TYPE UDT 19
VERSION : 0.0
  STRUCT
   A_SCLight : BOOL ;	//Screen light
   A_SCDark : BOOL ;	//Screen darkening
   A_KeyDisable : BOOL ;	//Key disable
   A_ClearCanAl : BOOL ;	//Clear cancel alarms
   A_ClearRecAl : BOOL ;	//Clear recall alarms
   f0_5 : BOOL ;
   f0_6 : BOOL ;
   A_ActWCS : BOOL ;	//Actual value in WCS 0=MCS
   A_PLCExtViewerReject : BOOL ;	//External viewer reject
   A_PLCExtViewerMode : BOOL ;	//External viewer mode
   f1_2 : BOOL ;
   f1_3 : BOOL ;
   f1_4 : BOOL ;
   f1_5 : BOOL ;
   f1_6 : BOOL ;
   f1_7 : BOOL ;
   A_1stError1 : WORD ;	//1st error HIGRAPH
   A_1stError2 : WORD ;	//1st error HIGRAPH
   A_ASpi1percent : BYTE ;	//Analog spindle 1:
   A_ASpi2percent : BYTE ;
   A_MCPChan : BYTE ;
   A_OEM1 : BOOL ;
   A_OEM2 : BOOL ;
   A_AToolMeas : BOOL ;	//AutoToolMeasure
   f9_3 : BOOL ;
   f9_4 : BOOL ;
   f9_5 : BOOL ;
   f9_6 : BOOL ;
   f9_7 : BOOL ;
   A_Hardkey : BYTE ;	//PLC Hardkeys
   f11 : BYTE ;	//Reserved for hardkeys
   f12_0 : BOOL ;
   f12_1 : BOOL ;
   A_COM2 : BOOL ;
   A_COM1 : BOOL ;
   A_V24stop : BOOL ;
   A_V24ext : BOOL ;
   A_V24off : BOOL ;
   A_V24on : BOOL ;
   A_TeachDisable : BOOL ;
   f13_1 : BOOL ;
   f13_2 : BOOL ;
   f13_3 : BOOL ;
   f13_4 : BOOL ;
   A_PPdeload : BOOL ;
   A_PPload : BOOL ;
   A_PPsel : BOOL ;
   A_V24Index1 : BYTE ;
   A_V24Index2 : BYTE ;
   A_V24NoFile1 : BYTE ;
   A_V24NoFile2 : BYTE ;
   A_res18 : BYTE ;
   A_res19 : BYTE ;	//Message counter
   f20_0 : BOOL ;
   E_SCDark : BOOL ;	//Screen darkening
   E_Cancel : BOOL ;	//Cancel
   E_CanCleared : BOOL ;	//Cancel alarms cleared
   E_RecCleared : BOOL ;	//Recall alarms cleared
   f20_5 : BOOL ;	//res. Language
   E_SimActiv : BOOL ;	//Simulation active
   E_ActWCS : BOOL ;	//Switchover MCS/WCS 0=MCS
   E_ActivWA : BYTE ;
   E_Chan : BYTE ;	//Channel displayed
   f23 : BYTE ;
   E_V24Err : BOOL ;
   E_V24OK : BOOL ;
   E_V24COM2 : BOOL ;
   E_V24COM1 : BOOL ;
   E_V24stop : BOOL ;
   E_V24ext : BOOL ;
   E_V24off : BOOL ;
   E_V24on : BOOL ;
   E_V24Error : BYTE ;	//V24: Error Byte
   E_res26_0 : BOOL ;	//Reserved
   E_PPOK : BOOL ;	//Part program status OK
   E_PPErr : BOOL ;	//Part program status Error
   E_PPAct : BOOL ;	//Part program status active
   f26_4 : BOOL ;	//Reserved
   E_PPdeload : BOOL ;	//Part program status deloading
   E_PPload : BOOL ;	//Part program status loading
   E_PPsel : BOOL ;	//Part program status selecting
   E_PPError : BYTE ;	//Part program status Error
   A_PictNo : INT ;
   A_PictOn : BOOL ;
   A_PictOff : BOOL ;
   f30_2 : BOOL ;
   f30_3 : BOOL ;
   f30_4 : BOOL ;
   f30_5 : BOOL ;
   f30_6 : BOOL ;
   f30_7 : BOOL ;
   E_PictOK : BOOL ;
   E_PictOn : BOOL ;
   E_PictAct : BOOL ;
   E_PictOff : BOOL ;
   E_PictErr : BOOL ;
   f31_5 : BOOL ;
   f31_6 : BOOL ;
   E_NotAct : BOOL ;
   A_FuncNo : BYTE ;
   A_Par1 : BYTE ;
   A_Par2 : BYTE ;
   A_Par3 : BYTE ;
   E_FuncErr : BYTE ;
   f37 : BYTE ;
   f38 : BYTE ;
   f39 : BYTE ;
   res40 : ARRAY  [0 .. 9 ] OF BYTE ;
   MMC2 : STRUCT
    A_SCLight : BOOL ;	//Screen light
    A_SCDark : BOOL ;	//Screen darkening
    A_KeyDisable : BOOL ;	//Key disable
    A_ClearCanAl : BOOL ;	//Clear cancel alarms
    A_ClearRecAl : BOOL ;	//Clear recall alarms
    f0_5 : BOOL ;
    f0_6 : BOOL ;
    A_ActWCS : BOOL ;	//Actual value in WCS 0=MCS
    A_1stError1 : WORD ;	//1st error HIGRAPH
    A_1stError2 : WORD ;	//1st error HIGRAPH
    A_ASpi1percent : BYTE ;	//Analog spindle 1:
    A_ASpi2percent : BYTE ;
    A_MCPChan : BYTE ;
    A_OEM1 : BOOL ;
    A_OEM2 : BOOL ;
    A_AToolMeas : BOOL ;	//AutoToolMeasure
    f9_3 : BOOL ;
    f9_4 : BOOL ;
    f9_5 : BOOL ;
    f9_6 : BOOL ;
    f9_7 : BOOL ;
    A_Hardkey : BYTE ;	//PLC Hardkeys
    f11 : BYTE ;	//Reserved for hardkeys
    f12_0 : BOOL ;
    f12_1 : BOOL ;
    A_COM2 : BOOL ;
    A_COM1 : BOOL ;
    A_V24stop : BOOL ;
    A_V24ext : BOOL ;
    A_V24off : BOOL ;
    A_V24on : BOOL ;
    f13_0 : BOOL ;
    f13_1 : BOOL ;
    f13_2 : BOOL ;
    f13_3 : BOOL ;
    f13_4 : BOOL ;
    A_PPdeload : BOOL ;
    A_PPload : BOOL ;
    A_PPsel : BOOL ;
    A_V24Index1 : BYTE ;
    A_V24Index2 : BYTE ;
    A_V24NoFile1 : BYTE ;
    A_V24NoFile2 : BYTE ;
    A_res18 : BYTE ;
    A_res19 : BYTE ;	//Message counter
    f20_0 : BOOL ;
    E_SCDark : BOOL ;	//Screen darkening
    E_Cancel : BOOL ;	//Cancel
    E_CanCleared : BOOL ;	//Cancel alarms cleared
    E_RecCleared : BOOL ;	//Recall alarms cleared
    f20_5 : BOOL ;	//res. Language
    E_SimActiv : BOOL ;	//Simulation active
    E_ActWCS : BOOL ;	//Switchover MCS/WCS 0=MCS
    E_ActivWA : BYTE ;
    E_Chan : BYTE ;	//Channel displayed
    f23 : BYTE ;
    E_V24Err : BOOL ;
    E_V24OK : BOOL ;
    E_V24COM2 : BOOL ;
    E_V24COM1 : BOOL ;
    E_V24stop : BOOL ;
    E_V24ext : BOOL ;
    E_V24off : BOOL ;
    E_V24on : BOOL ;
    E_V24Error : BYTE ;	//V24: Error Byte
    E_res26_0 : BOOL ;	//Reserved
    E_PPOK : BOOL ;	//Part program status OK
    E_PPErr : BOOL ;	//Part program status Error
    E_PPAct : BOOL ;	//Part program status active
    f26_4 : BOOL ;	//Reserved
    E_PPdeload : BOOL ;	//Part program status deloading
    E_PPload : BOOL ;	//Part program status loading
    E_PPsel : BOOL ;	//Part program status selecting
    E_PPError : BYTE ;	//Part program status Error
    A_PictNo : INT ;
    A_PictOn : BOOL ;
    A_PictOff : BOOL ;
    f30_2 : BOOL ;
    f30_3 : BOOL ;
    f30_4 : BOOL ;
    f30_5 : BOOL ;
    f30_6 : BOOL ;
    f30_7 : BOOL ;
    E_PictOK : BOOL ;
    E_PictOn : BOOL ;
    E_PictAct : BOOL ;
    E_PictOff : BOOL ;
    E_PictErr : BOOL ;
    f31_5 : BOOL ;
    f31_6 : BOOL ;
    E_NotAct : BOOL ;
    A_FuncNo : BYTE ;
    A_Par1 : BYTE ;
    A_Par2 : BYTE ;
    A_Par3 : BYTE ;
    E_FuncErr : BYTE ;
    f37 : BYTE ;
    f38 : BYTE ;
    f39 : BYTE ;
    res40 : ARRAY  [0 .. 9 ] OF BYTE ;
   END_STRUCT ;	//M to N
   ONL_REQUEST : WORD ;
   ONL_CONFIRM : WORD ;
   PAR_CLIENT_IDENT : WORD ;
   PAR_MMC_TYP : BYTE ;
   PAR_MSTT_ADR : BYTE ;
   PAR_STATUS : BYTE ;
   PAR_Z_INFO : BYTE ;
   MtoNAlive : WORD ;
   f112 : BYTE ;
   ParOpKeyAdr : BYTE ;
   ParTcuIndex : BYTE ;
   f115 : BYTE ;
   Tcu1KeyAdr : BYTE ;
   Tcu2KeyAdr : BYTE ;
   Tcu1Index : BYTE ;
   Tcu2Index : BYTE ;
   MMC1_CLIENT_IDENT : WORD ;
   MMC1_TYP : BYTE ;
   MMC1_MSTT_ADR : BYTE ;
   MMC1_STATUS : BYTE ;
   MMC1_Z_INFO : BYTE ;
   MMC1_SHIFT_LOCK : BOOL ;
   MMC1_MSTT_SHIFT_LOCK : BOOL ;
   MMC1_ACTIVE_REQ : BOOL ;
   MMC1_ACTIVE_PERM : BOOL ;
   MMC1_ACTIVE_CHANGED : BOOL ;
   MMC1_CHANGED_DENIED : BOOL ;
   MMC1_TCU_SHIFT_LOCK : BOOL ;
   f127 : BYTE ;
   MMC1_TRANS_DB : WORD ;
   MMC2_CLIENT_IDENT : WORD ;
   MMC2_TYP : BYTE ;
   MMC2_MSTT_ADR : BYTE ;
   MMC2_STATUS : BYTE ;
   MMC2_Z_INFO : BYTE ;
   MMC2_SHIFT_LOCK : BOOL ;
   MMC2_MSTT_SHIFT_LOCK : BOOL ;
   MMC2_ACTIVE_REQ : BOOL ;
   MMC2_ACTIVE_PERM : BOOL ;
   MMC2_ACTIVE_CHANGED : BOOL ;
   MMC2_CHANGED_DENIED : BOOL ;
   MMC2_TCU_SHIFT_LOCK : BOOL ;
   f137 : BYTE ;
   MMC2_TRANS_DB : WORD ;
   A_Subtype : INT ;	//for Codecarrier Input from PLC
   A_Duplo : INT ;
   A_Ident : STRING  [32 ];
   A_Tnumber : INT ;
   A_MagazinePlace : INT ;
   A_MagazinePlaceType : INT ;
   A_ToolSize_Upper : BYTE ;
   A_ToolSize_Down : BYTE ;
   A_ToolSize_Left : BYTE ;
   A_ToolSize_Right : BYTE ;
   A_Channel : BYTE ;
   A_LoadingPlace : BYTE ;
   A_Magazine : INT ;
   A_Unit : BYTE ;
   A_NCU_Index : BYTE ;
   A_FileIndex : INT ;
   A_ActiveEnable : BOOL ;
   A_Override : BOOL ;
   A_LoadTool : BOOL ;
   A_DeleteTool : BOOL ;
   E_Subtype : INT ;	//for Codecarrier Output to PLC
   E_Duplo : INT ;
   E_Ident : STRING  [32 ];
   E_Tnumber : INT ;
   E_ToolState : INT ;
   E_MagazinePlaceType : INT ;
   E_ToolSize_Upper : BYTE ;
   E_ToolSize_Down : BYTE ;
   E_ToolSize_Left : BYTE ;
   E_ToolSize_Right : BYTE ;
   E_Magazine : INT ;
   E_MagazinePlace : INT ;
   A_ReqMMC1 : BOOL ;	//for Codecarrier Request MMC-Interface1
   A_ReqMMC2 : BOOL ;	//for Codecarrier Request MMC-Interface2
   A_K_Code : BYTE ;
   E_Done : BOOL ;
   E_Error : BOOL ;
   E_Active : BOOL ;	// CodeCarrierReadEnable : BOOL;
// CodeCarrierWriteEnable : BOOL;
   E_K_CodeError : BYTE ;	//Identify for Error_Code
   E_Error_Code : INT ;
   E_Req : BOOL ;	//for Positioning
   f257 : BYTE ;
   A_Done : BOOL ;
   A_Error : BOOL ;
   A_Active : BOOL ;
   f258_3 : BOOL ;
   f258_4 : BOOL ;
   f258_5 : BOOL ;
   f258_6 : BOOL ;
   f258_7 : BOOL ;
   E_TDC_Read : BOOL ;
   E_TDC_Write : BOOL ;
   E_TDC_Cancel : BOOL ;
   A_Error_Code : INT ;
   E_PMagazine : INT ;
   E_PMagazinePlace : INT ;
   E_PTnumber : INT ;	//TPM-Data
   A_TPMStatus : INT ;
   A_TPMCounter : ARRAY  [1 .. 32 ] OF DINT ;
   A_HWeelSimOvr : BYTE ;
   f399 : BYTE ;
   A_SimOvr : INT ;
  END_STRUCT ;	
END_TYPE

TYPE UDT 21
VERSION : 0.0
  STRUCT
   f0_0 : BOOL ;
   f0_1 : BOOL ;
   f0_2 : BOOL ;
   A_DRF : BOOL ;	//Activate DRF
   A_SBL : BOOL ;	//Activate single block
   A_M01 : BOOL ;	//Activate M01
   A_DRY : BOOL ;	//Activate dry run feedrate
   f0_7 : BOOL ;
   A_Ref : BOOL ;	//Activate referencing
   A_ProtZone : BOOL ;	//Enable protection zones
   A_SynOff : BOOL ;	//Synchronous action off
   A_TM_TimOut : BOOL ;	//Activate time-out (TM)
   A_CLC_Stop : BOOL ;	//CLC stop
   A_CLC_OR : BOOL ;	//CLC override
   A_PLC_ActCompl : BOOL ;	//PLC action complete
   A_ProgTest : BOOL ;	//Activate program test
   A_SKP0 : BOOL ;	//Activate skip block \0
   A_SKP1 : BOOL ;	//Activate skip block \1
   A_SKP2 : BOOL ;	//Activate skip block \2
   A_SKP3 : BOOL ;	//Activate skip block \3
   A_SKP4 : BOOL ;	//Activate skip block \4
   A_SKP5 : BOOL ;	//Activate skip block \5
   A_SKP6 : BOOL ;	//Activate skip block \6
   A_SKP7 : BOOL ;	//Activate skip block \7
   A_StrokEnab : BOOL ;	//Stroke enable
   A_ManStrokEnab : BOOL ;	//Manual stroke enable
   A_StrokSup : BOOL ;	//Stroke suppression
   A_StrokDelayed : BOOL ;	//Stroke delayed
   A_StrokStop : BOOL ;	//Stroke not operating
   A_ManRelStroke2 : BOOL ;	// Manual release of stroke 2
   A3_6 : BOOL ;
   A3_7 : BOOL ;
   A_FD_OR : BYTE ;	//Feedrate override
   A_RT_OR : BYTE ;	//Rapid traverse override
   A_FDdisable : BOOL ;	//Feed disable
   A_RIdisable : BOOL ;	//Read-in disable
   A_DeleteDTG : BOOL ;	//Delete distance to go
   A_SP_Clear : BOOL ;	//Clear SP repetitions
   A_ProgAbort : BOOL ;	//Program level abort
   A_F_Limit : BOOL ;	//Tool path feedrate limitation
   A_RT_ORA : BOOL ;	//Rapid traverse override active
   A_FD_ORA : BOOL ;	//Feedrate override active
   A_NCStartDisabl : BOOL ;	//NC start disable
   A_NCStart : BOOL ;	//NC start
   A_NCStopBlock : BOOL ;	//NC stop at block limit
   A_NCStop : BOOL ;	//NC stop
   A_NCStopASp : BOOL ;	//NC stop axes plus spindle
   A_SuppStartLock : BOOL ;	// Suppress Start Lock
   f7_6 : BOOL ;
   A_Reset : BOOL ;	//Reset
   A_MRP : ARRAY  [1 .. 10 ] OF BOOL ;	//Activate machine-related protection area [1..10]
   A_CSP : ARRAY  [1 .. 10 ] OF BOOL ;	//Activate channel-specific protection area [1..10]
   A_Geo : ARRAY  [1 .. 3 ] OF STRUCT 	//Control signals for geometry axis [1..3]
    HW1 : BOOL ;	//Activate handwheel 1
    HW2 : BOOL ;	//Activate handwheel 2
    HW3 : BOOL ;	//Activate handwheel 3
    FDStop : BOOL ;	//Feed stop
    Disabl : BOOL ;	//Traversing key disable
    RapidTrOR : BOOL ;	//Rapid traverse override
    Minus : BOOL ;	//Traversing key minus
    Plus : BOOL ;	//Traversing key plus
    INC1 : BOOL ;	//INC 1
    INC10 : BOOL ;	//INC 10
    INC100 : BOOL ;	//INC 100
    INC1000 : BOOL ;	//INC 1000
    INC10000 : BOOL ;	//INC 10000
    INCVar : BOOL ;	//INC variable
    OEM : BYTE ;	//OEM signals
    InvHWDirOfRot : BOOL ;	// Inverting handwheel direction of rotation
    f3_1 : BOOL ;
    f3_2 : BOOL ;
    f3_3 : BOOL ;
    f3_4 : BOOL ;
    f3_5 : BOOL ;
    f3_6 : BOOL ;
    f3_7 : BOOL ;
   END_STRUCT ;
   f24_0 : BOOL ;
   f24_1 : BOOL ;
   f24_2 : BOOL ;
   E_MMC_DRF : BOOL ;	//MMC DRF selected
   f24_4 : BOOL ;
   E_MMC_M01 : BOOL ;	//MMC M01 selected
   E_MMC_DRY : BOOL ;	//MMC Dry run feedrate selected
   f24_7 : BOOL ;
   E_MMC_REPOSPM_0 : BOOL ;	//MMC REPOSPATHMODE 0
   E_MMC_REPOSPM_1 : BOOL ;	//MMC REPOSPATHMODE 1
   E_MMC_REPOSPM_2 : BOOL ;	//MMC REPOSPATHMODE 2
   E_MMC_FD_OR4RT_OR : BOOL ;	//MMC Feedrate override for rapid traverse selected
   E_MMC_REPOSMode : BOOL ;	//MMC REPOS MODE EDGE
   f25_5 : BOOL ;
   f25_6 : BOOL ;
   E_MMC_ProgTest : BOOL ;	//Program test selected
   E_MMC_SKP0 : BOOL ;	//MMC skip block selected \0
   E_MMC_SKP1 : BOOL ;	//MMC skip block selected \1
   E_MMC_SKP2 : BOOL ;	//MMC skip block selected \2
   E_MMC_SKP3 : BOOL ;	//MMC skip block selected \3
   E_MMC_SKP4 : BOOL ;	//MMC skip block selected \4
   E_MMC_SKP5 : BOOL ;	//MMC skip block selected \5
   E_MMC_SKP6 : BOOL ;	//MMC skip block selected \6
   E_MMC_SKP7 : BOOL ;	//MMC skip block selected \7
   E_MMC_SKP8 : BOOL ;	//MMC skip block selected \8
   E_MMC_SKP9 : BOOL ;	//MMC skip block selected \9
   f27_2 : BOOL ;
   f27_3 : BOOL ;
   f27_4 : BOOL ;
   f27_5 : BOOL ;
   f27_6 : BOOL ;
   f27_7 : BOOL ;
   A_OEM : BYTE ;
   A_FixedFD1 : BOOL ;	//Fixed feeds
   A_FixedFD2 : BOOL ;
   A_FixedFD3 : BOOL ;
   A_FixedFD4 : BOOL ;
   A_PTP_Travel : BOOL ;	//Activate PTP travel
   A_DisablWP_Counter : BOOL ;	//Disable workpiece counter
   A_DisablWearMon : BOOL ;	//Disable wear monitoring
   A_DontDisablTool : BOOL ;	//Do not disable tool
   A_ContHW1 : BOOL ;	//Activate contour handwheels
   A_ContHW2 : BOOL ;
   A_ContHW3 : BOOL ;
   A_ContHWsim : BOOL ;	//Simulated contour handwheel on
   A_ContHWneg : BOOL ;	//Contour handwheel neg. route
   A_NCKrelatedM01 : BOOL ;	// Activate NCK-related M01
   f30_6 : BOOL ;
   A_NoToolChangeCmd : BOOL ;	// No tool change commands
   A_REPOSPM_0 : BOOL ;	//REPOSPATHMODE 0
   A_REPOSPM_1 : BOOL ;	//REPOSPATHMODE 1
   A_REPOSPM_2 : BOOL ;	//REPOSPATHMODE 2
   f31_3 : BOOL ;
   A_REPOSMode : BOOL ;	//REPOS MODE EDGE
   A_InvCHWDirOfRot : BOOL ;	// Inverting contour handwheel direction of rotation
   A_SKP8 : BOOL ;	//Activate skip block \8
   A_SKP9 : BOOL ;	//Activate skip block \9
   E_ExecExtern : BOOL ;	//Execution from external source active
   f32_1 : BOOL ;
   f32_2 : BOOL ;
   E_ActBlock : BOOL ;	//Action block active
   E_BegBlock : BOOL ;	//Approach block active
   E_M01 : BOOL ;	//M0/M1 active
   E_LastActBlock : BOOL ;	//Last action block active
   f32_7 : BOOL ;
   E_Ref : BOOL ;	//Referencing active
   E_OrieToolholder : BOOL ;	// Orientable toolholder active
   E_RevFD : BOOL ;	//Revolutional feedrate active
   E_HWOverlay : BOOL ;	//Handwheel overlay active
   E_BlockSearch : BOOL ;	//Block search active
   E_M30 : BOOL ;	//M2/M30 active
   E_Transform : BOOL ;	//Transformation active
   E_ProgTest : BOOL ;	//Program test active
   E_OEMChan : BYTE ;	//OEM channel signals feedback
   E_ProgRunn : BOOL ;	//Program running
   E_ProgWait : BOOL ;	//Program waiting
   E_ProgStop : BOOL ;	//Program stopped
   E_ProgInterrupt : BOOL ;	//Program interrupted
   E_ProgrAborted : BOOL ;	//Program aborted
   E_ChanActive : BOOL ;	//Channel active
   E_ChanInterrupt : BOOL ;	//Channel interrupted
   E_ChanReset : BOOL ;	//Channel reset
   E_StartReq : BOOL ;	//Start request
   E_StopReq : BOOL ;	//Stop request
   E_AxesRef : BOOL ;	//All axes referenced
   E_AxesStop : BOOL ;	//All axes stationary
   E_IR_Activ : BOOL ;	//Interrupt processing active
   E_ChanRO : BOOL ;	//Channel ready for operation
   E_NCKalarmChan : BOOL ;	//Channel-specific NCK alarm present
   E_NCKalarmStop : BOOL ;	//NCK alarm with processing stop present
   E_CHW1 : BOOL ;	//Contour handwheel 1 on
   E_CHW2 : BOOL ;	//Contour handwheel 2 on
   E_CHW3 : BOOL ;	//Contour handwheel 3 on
   E_CLC : BOOL ;	//CLC active
   E_CLCStopLL : BOOL ;	//CLC stopped lower limit
   E_CLCStopUL : BOOL ;	//CLC stopped upper limit
   E_RIEnabIgnored : BOOL ;	//Read-in enable is ignored
   E_StopBlkEndSBLsuppr : BOOL ;	//Stop at block end with SBL is suppressed
   E_StrokeEA : BOOL ;	//Stroke enable active
   E_AcknManStrokEnab : BOOL ;	//Acknowledgement manual stroke enable
   f38_2 : BOOL ;
   f38_3 : BOOL ;
   f38_4 : BOOL ;
   f38_5 : BOOL ;
   f38_6 : BOOL ;
   f38_7 : BOOL ;
   E_ProtZoneNOK : BOOL ;	//Protection zones not guaranteed
   f39_1 : BOOL ;
   f39_2 : BOOL ;
   f39_3 : BOOL ;
   f39_4 : BOOL ;
   E_InvCHWDirOfRot : BOOL ;	// Contour handwheel direction of rotation invert actively
   f39_6 : BOOL ;
   f39_7 : BOOL ;
   E_Geo : ARRAY  [1 .. 3 ] OF STRUCT 	//Status signals of geometry axis [1..3]
    HW1 : BOOL ;	//Handwheel 1 active
    HW2 : BOOL ;	//Handwheel 2 active
    HW3 : BOOL ;	//Handwheel 3 active
    f0_3 : BOOL ;
    TReqMinus : BOOL ;	// Travel requests minus
    TReqPlus : BOOL ;	// Travel requests plus
    TCMinus : BOOL ;	//Traverse command minus
    TCPlus : BOOL ;	//Traverse command plus
    INC1 : BOOL ;	//INC 1 active
    INC10 : BOOL ;	//INC 10 active
    INC100 : BOOL ;	//INC 100 active
    INC1000 : BOOL ;	//INC 1000 active
    INC10000 : BOOL ;	//INC 10000 active
    INCVar : BOOL ;	//INC variable active
    OEM : BYTE ;	//OEM signals
    InvHWDirOfRot : BOOL ;	// Handwheel direction of rotation invert actively
    f3_1 : BOOL ;
    f3_2 : BOOL ;
    f3_3 : BOOL ;
    f3_4 : BOOL ;
    f3_5 : BOOL ;
    f3_6 : BOOL ;
    f3_7 : BOOL ;
    f4 : BYTE ;
   END_STRUCT ;
   M1Change : BOOL ;	//M function 1 change
   M2Change : BOOL ;	//M function 2 change
   M3Change : BOOL ;	//M function 3 change
   M4Change : BOOL ;	//M function 4 change
   M5Change : BOOL ;	//M function 5 change
   f58_5 : BOOL ;
   f58_6 : BOOL ;
   f58_7 : BOOL ;
   M1NDec : BOOL ;	//M function 1 not decoded
   M2NDec : BOOL ;	//M function 2 not decoded
   M3NDec : BOOL ;	//M function 3 not decoded
   M4NDec : BOOL ;	//M function 4 not decoded
   M5NDec : BOOL ;	//M function 5 not decoded
   f59_5 : BOOL ;
   f59_6 : BOOL ;
   f59_7 : BOOL ;
   S1Change : BOOL ;	//S function 1 change
   S2Change : BOOL ;	//S function 2 change
   S3Change : BOOL ;	//S function 3 change
   f60_3 : BOOL ;
   S1Quick : BOOL ;	//S function 1 quick
   S2Quick : BOOL ;	//S function 2 quick
   S3Quick : BOOL ;	//S function 3 quick
   f60_7 : BOOL ;
   T1Change : BOOL ;	//T function 1 change
   T2Change : BOOL ;	//T function 2 change
   T3Change : BOOL ;	//T function 3 change
   f61_3 : BOOL ;
   T1Quick : BOOL ;	//T function 1 quick
   T2Quick : BOOL ;	//T function 2 quick
   T3Quick : BOOL ;	//T function 3 quick
   f61_7 : BOOL ;
   D1Change : BOOL ;	//D function 1 change
   D2Change : BOOL ;	//D function 2 change
   D3Change : BOOL ;	//D function 3 change
   f62_3 : BOOL ;
   D1Quick : BOOL ;	//D function 1 quick
   D2Quick : BOOL ;	//D function 2 quick
   D3Quick : BOOL ;	//D function 3 quick
   f62_7 : BOOL ;
   EChange : BOOL ;	//E function change
   f63_1 : BOOL ;
   f63_2 : BOOL ;
   f63_3 : BOOL ;
   EQuick : BOOL ;	//E function quick
   f63_5 : BOOL ;
   f63_6 : BOOL ;
   f63_7 : BOOL ;
   H1Change : BOOL ;	//H function 1 change
   H2Change : BOOL ;	//H function 2 change
   H3Change : BOOL ;	//H function 3 change
   f64_3 : BOOL ;
   H1Quick : BOOL ;	//H function 1 quick
   H2Quick : BOOL ;	//H function 2 quick
   H3Quick : BOOL ;	//H function 3 quick
   f64_7 : BOOL ;
   F1Change : BOOL ;	//F function 1 change
   F2Change : BOOL ;	//F function 2 change
   F3Change : BOOL ;	//F function 3 change
   F4Change : BOOL ;	//F function 4 change
   F5Change : BOOL ;	//F function 5 change
   F6Change : BOOL ;	//F function 6 change
   f65_6 : BOOL ;
   f65_7 : BOOL ;
   M1Quick : BOOL ;	//M function 1 quick
   M2Quick : BOOL ;	//M function 2 quick
   M3Quick : BOOL ;	//M function 3 quick
   M4Quick : BOOL ;	//M function 4 quick
   M5Quick : BOOL ;	//M function 5 quick
   f66_5 : BOOL ;
   f66_6 : BOOL ;
   f66_7 : BOOL ;
   F1Quick : BOOL ;	//F function 1 quick
   F2Quick : BOOL ;	//F function 2 quick
   F3Quick : BOOL ;	//F function 3 quick
   F4Quick : BOOL ;	//F function 4 quick
   F5Quick : BOOL ;	//F function 5 quick
   F6Quick : BOOL ;	//F function 6 quick
   f67_6 : BOOL ;
   f67_7 : BOOL ;
   ExtM1 : INT ;	//Extended address M function 1 (16 bit INT)
   M1 : DINT ;	//M function 1 (DInt)
   ExtM2 : INT ;	//Extended address M function 1 (16 bit INT)
   M2 : DINT ;	//M function 2 (DInt)
   ExtM3 : INT ;	//Extended address M function 1 (16 bit INT)
   M3 : DINT ;	//M function 3 (DInt)
   ExtM4 : INT ;	//Extended address M function 1 (16 bit INT)
   M4 : DINT ;	//M function 4 (DInt)
   ExtM5 : INT ;	//Extended address M function 1 (16 bit INT)
   M5 : DINT ;	//M function 5 (DInt)
   ExtS1 : INT ;	//Extended address S function 1 (16 bit INT)
   S1 : REAL ;	//S function 1 (REAL)
   ExtS2 : INT ;	//Extended address S function 2 (16 bit INT)
   S2 : REAL ;	//S function 2 (REAL)
   ExtS3 : INT ;	//Extended address S function 3 (16 bit INT)
   S3 : REAL ;	//S function 3 (REAL)
   ExtT1 : INT ;	//Extended address T function 1 (16 bit INT)
//T : DINT; //T function (DInt)
//f122 :
   T1 : INT ;	//T function 1 (INT)
   ExtT2 : INT ;	//Extended address T function 2 (16 bit INT)
   T2 : INT ;	//T function 2 (INT)
   ExtT3 : INT ;	//Extended address T function 3 (16 bit INT)
   T3 : INT ;	//T function 3 (INT)
   ExtD1 : BYTE ;	//Extended address D function 1 (8 bit INT)
//D : INT;
//f132 : INT;   //Change in ca
   D1 : BYTE ;	//D function 1 (8 bit INT)
   ExtD2 : BYTE ;	//Extended address D function 2 (8 bit INT)
   D2 : BYTE ;	//D function 2 (8 bit INT)
   ExtD3 : BYTE ;	//Extended address D function 3 (8 bit INT)
   D3 : BYTE ;	//D function 3 (8 bit INT)
   ExtE : INT ;	//Extended address E function 3 (16 bit INT)
   E : REAL ;	//E function (REAL)
   ExtH1 : INT ;	//Extended address H function 1 (16 bit INT)
   H1 : REAL ;	//H function 1 (REAL)
   ExtH2 : INT ;	//Extended address H function 2 (16 bit INT)
   H2 : REAL ;	//H function 2 (REAL)
   ExtH3 : INT ;	//Extended address H function 3 (16 bit INT)
   H3 : REAL ;	//H function 3 (REAL)
   ExtF1 : INT ;	//Extended address F function 1 (16 bit INT)
   F1 : REAL ;	//F function 1 (REAL)
   ExtF2 : INT ;	//Extended address F function 2 (16 bit INT)
   F2 : REAL ;	//F function 2 (REAL)
   ExtF3 : INT ;	//Extended address F function 3 (16 bit INT)
   F3 : REAL ;	//F function 3 (REAL)
   ExtF4 : INT ;	//Extended address F function 4 (16 bit INT)
   F4 : REAL ;	//F function 4 (REAL)
   ExtF5 : INT ;	//Extended address F function 5 (16 bit INT)
   F5 : REAL ;	//F function 5 (REAL)
   ExtF6 : INT ;	//Extended address F function 6 (16 bit INT)
   F6 : REAL ;	//F function 6 (REAL)
   MDyn : ARRAY  [0 .. 99 ] OF BOOL ;	//Dynamic M functions [0..99]
   GAct : ARRAY  [1 .. 64 ] OF BYTE ;	//Active G function of group [1..64]
   E_MRPactivated : ARRAY  [1 .. 10 ] OF BOOL ;	//Machine-related protection area [1..10] preactivated
   E_CSPactivated : ARRAY  [1 .. 10 ] OF BOOL ;	//Channel-specific protection area [1..10] preactivated
   E_MRPViolated : ARRAY  [1 .. 10 ] OF BOOL ;	//Machine-related protection area [1..10] violated
   E_CSPViolated : ARRAY  [1 .. 10 ] OF BOOL ;	//Channel-specific protection area [1..10] violated
//from P4 on
   A_Str_DNo : BOOL ;	//Request of D number to NCK
   A_Str_Synon : BOOL ;	//Request of syn.action to NCK
   f_280_2 : BOOL ;
   f_280_3 : BOOL ;
   f_280_4 : BOOL ;
   f_280_5 : BOOL ;
   f_280_6 : BOOL ;
   f_280_7 : BOOL ;
   f_281_0 : BOOL ;
   A_Str_Synfrom : BOOL ;	//Request syn.action from NCK
   f_281_2 : BOOL ;
   f_281_3 : BOOL ;
   f_281_4 : BOOL ;
   f_281_5 : BOOL ;
   f_281_6 : BOOL ;
   f_281_7 : BOOL ;
   A_D1 : INT ;	//Assignment D1
   A_D2 : INT ;	//Assignment D2
   A_D3 : INT ;	//Assignment D3
   A_D4 : INT ;	//Assignment D4
   A_D5 : INT ;	//Assignment D5
   A_D6 : INT ;	//Assignment D6
   A_D7 : INT ;	//Assignment D7
   A_D8 : INT ;	//Assignment D8
   A_D9 : INT ;	//Assignment D9
   A_SynDisabl : ARRAY  [1 .. 64 ] OF BOOL ;	//Disable synchronous actions
   E_SynDisabled : ARRAY  [1 .. 64 ] OF BOOL ;	//Synchronous actions disabled
   E_G00 : BOOL ;	//Active G functions
   f316_1 : BOOL ;
   f316_2 : BOOL ;
   f316_3 : BOOL ;
   f316_4 : BOOL ;
   f316_5 : BOOL ;
   f316_6 : BOOL ;
   f316_7 : BOOL ;
   E_ExtLang : BOOL ;	// External language mode active
   E_WS_Setp : BOOL ;	// Workpiece setpoint reached
   f317_2 : BOOL ;
   f317_3 : BOOL ;
   f317_4 : BOOL ;
   E_DriveTest : BOOL ;	// Travel request drive test
   E_PTP_Travel : BOOL ;	//PTP travel active
   E_ToolMissing : BOOL ;	//Tool missing
   E_ASUP_Stop : BOOL ;	// ASUP stopped
   E_SearchAct : BOOL ;	// Search active
   E_TOFF : BOOL ;	// TOFF active
   E_TOFFmovem : BOOL ;	// TOFF movement active
   E_StopDelayed : BOOL ;	// Stop delayed
   E_AssM01 : BOOL ;	// Associated M01 active
   E_DRY : BOOL ;	// Dry-run feedrate active
   E_Overstore : BOOL ;	// Overstore active
   E_REPOS_EdgeAckn : BOOL ;	// REPOS MODE EDGE ACKN
   E_REPOS_PMode0 : BOOL ;	// Repos Path Mode Ackn 0
   E_REPOS_PMode1 : BOOL ;	// Repos Path Mode Ackn 0
   E_REPOS_PMode2 : BOOL ;	// Repos Path Mode Ackn 2
   E_DelayFTS : BOOL ;	// Delay FTS
   E_REPOS_DEFERRA : BOOL ;	// Repos DEFERRA L Chan
   E_Stop_NoDelayR : BOOL ;	// Stop-delayrange not activated
   E_NoToolChangeCmd : BOOL ;	// No tool change command active
   A_Ori : ARRAY  [1 .. 3 ] OF STRUCT 	//Control signals for orientation axes [1..3]
    HW_Bit0 : BOOL ;	//Activate handwheel Bit value coding
    HW_Bit1 : BOOL ;	//Activate handwheel Bit value coding
    HW_Bit2 : BOOL ;	//Activate handwheel Bit value coding
    FDStop : BOOL ;	//Feed stop
    Disabl : BOOL ;	//Traversing key disable
    RapidTrOR : BOOL ;	//Rapid traverse override
    Minus : BOOL ;	//Traversing key minus
    Plus : BOOL ;	//Traversing key plus
    INC1 : BOOL ;	//INC 1 active
    INC10 : BOOL ;	//INC 10 active
    INC100 : BOOL ;	//INC 100 active
    INC1000 : BOOL ;	//INC 1000 active
    INC10000 : BOOL ;	//INC 10000 active
    INCVar : BOOL ;	//INC variable active
    OEM : BYTE ;	//OEM signals
    InvHWDirOfRot : BOOL ;	// Inverting handwheel direction of rotation
    f3_1 : BOOL ;
    f3_2 : BOOL ;
    f3_3 : BOOL ;
    f3_4 : BOOL ;
    f3_5 : BOOL ;
    f3_6 : BOOL ;
    f3_7 : BOOL ;
   END_STRUCT ;
   E_Ori : ARRAY  [1 .. 3 ] OF STRUCT 	//Control signals for orientation axes [1..3]
    HW_Bit0 : BOOL ;	//Activate handwheel Bit value coding
    HW_Bit1 : BOOL ;	//Activate handwheel Bit value coding
    HW_Bit2 : BOOL ;	//Activate handwheel Bit value coding
    f0_3 : BOOL ;
    TReqMinus : BOOL ;	// Travel requests minus
    TReqPlus : BOOL ;	// Travel requests plus
    Minus : BOOL ;	//Traversing key minus
    Plus : BOOL ;	//Traversing key plus
    INC1 : BOOL ;	//INC 1 active
    INC10 : BOOL ;	//INC 10 active
    INC100 : BOOL ;	//INC 100 active
    INC1000 : BOOL ;	//INC 1000 active
    INC10000 : BOOL ;	//INC 10000 active
    INCVar : BOOL ;	//INC variable active
    OEM : BYTE ;	//OEM signals
    InvHWDirOfRot : BOOL ;	// Handwheel direction of rotation invert actively
    f3_1 : BOOL ;
    f3_2 : BOOL ;
    f3_3 : BOOL ;
    f3_4 : BOOL ;
    f3_5 : BOOL ;
    f3_6 : BOOL ;
    f3_7 : BOOL ;
   END_STRUCT ;
   E_T_PrewarnLimit : BOOL ;	//Tool prewarn limit reached
   E_T_Limit : BOOL ;	//Tool limit reached
   E_NewReplT : BOOL ;	//Transition to new replacement tool
   E_LastReplT : BOOL ;	//last replacement tool of the tool group
   f344_4 : BOOL ;
   f344_5 : BOOL ;
   f344_6 : BOOL ;
   f344_7 : BOOL ;
   f345 : BYTE ;
   f346 : BYTE ;
   f347 : BYTE ;
   E_T_NoPrewarnLimit : DINT ;	//T number for tool prewarn limit
   E_T_NoLimit : DINT ;	//T number for tool limit
   E_NewReplT_No : DINT ;	//T number of the new replacement tool
   E_LastReplT_No : DINT ;	//T number of the last replacement tool
   E_Cycle_Sig : ARRAY  [0 .. 15 ] OF BOOL ;	//Cycles Input Signals
   A_Cycle_Sig : ARRAY  [0 .. 15 ] OF BOOL ;	//Cycles Output Signals
   E_OEM_TechnoSig : ARRAY  [0 .. 31 ] OF BOOL ;	//OEM Techno Input Signals
   A_OEM_TechnoSig : ARRAY  [0 .. 31 ] OF BOOL ;	//OEM Techno Output Signals
   ProgEventDispl : BYTE ;	// ProgEventDisplay
   E_CollCheckStop : BOOL ;	// Stop of Collision Check
   E_StopCondition : BOOL ;	// Stop Condition
   f377_2 : BOOL ;
   f377_3 : BOOL ;
   f377_4 : BOOL ;
   f377_5 : BOOL ;
   f377_6 : BOOL ;
   f377_7 : BOOL ;
   E_AnyAsup : BOOL ;	// AnyASUP activ
   E_SilentAsup : BOOL ;	// Silent ASUP activ
   f378_2 : BOOL ;
   f378_3 : BOOL ;
   f378_4 : BOOL ;
   f378_5 : BOOL ;
   f378_6 : BOOL ;
   f378_7 : BOOL ;
   f379 : BYTE ;
   f380 : ARRAY  [0 .. 31 ] OF BOOL ;	//Reserved
   A_ProgJump : BOOL ;	// control program jump
   f384_1 : BOOL ;
   f384_2 : BOOL ;
   f384_3 : BOOL ;
   f384_4 : BOOL ;
   f384_5 : BOOL ;
   f384_6 : BOOL ;
   f384_7 : BOOL ;
   f385 : BYTE ;
   f386 : WORD ;
   E_TransfoNo : BYTE ;	// active Transformation No.
   f389 : BYTE ;
   f390 : WORD ;
  END_STRUCT ;	
END_TYPE

TYPE UDT 31
VERSION : 0.0
  STRUCT
   A_FD_OR : BYTE ;	//Feedrate override
   A_DriveEnable : BOOL ;	//Drive test movement enable
   A_AckFixedStop : BOOL ;	//Acknowledge fixed stop reached
   A_SensorFixedStop : BOOL ;	//Sensor fixed stop
   A_ASpDisable : BOOL ;	//Axis/spindle disable
   A_Follow_upMode : BOOL ;	//Follow-up mode
   A_PosMeas1 : BOOL ;	//Position measuring system 1
   A_PosMeas2 : BOOL ;	//Position measuring system 2
   A_ORactive : BOOL ;	//Override active
   A_SWCam : BOOL ;	//SW cam activation
   A_ContrEnable : BOOL ;	//Controller enable
   A_DelDTGSpReset : BOOL ;	//Delete distance to go/Spindle-Reset
   A_Clamp : BOOL ;	//Clamping in progress
   A_RefVal1 : BOOL ;	//Reference point value 1
   A_RefVal2 : BOOL ;	//Reference point value 2
   A_RefVal3 : BOOL ;	//Reference point value 3
   A_RefVal4 : BOOL ;	//Reference point value 4
   A_ExtZO : BOOL ;	//Import external ZO
   A_EnabTravFixedStop : BOOL ;	//Enable travel to fixed stop
   A_FixedFD1 : BOOL ;	//Activate fixed feed 1
   A_FixedFD2 : BOOL ;	//Activate fixed feed 2
   A_FixedFD3 : BOOL ;	//Activate fixed feed 3
   A_FixedFD4 : BOOL ;	//Activate fixed feed 4
   A_VelocSpeedLimit : BOOL ;	//Velocity/spindle speed limitation
   A_PrgtestAxRel : BOOL ;	// Program test axis/spindle release
   A_HW1 : BOOL ;	//Activate handwheel 1
   A_HW2 : BOOL ;	//Activate handwheel 2
   A_HW3 : BOOL ;	//Activate handwheel 3
   A_FDSpStop : BOOL ;	//Feed stop/spindle stop
   A_Disable : BOOL ;	//Traversing key disable
   A_RapidTrOR : BOOL ;	//Rapid traverse override
   A_Minus : BOOL ;	//Traversing key minus
   A_Plus : BOOL ;	//Traversing key plus
   A_INC1 : BOOL ;	//INC1
   A_INC10 : BOOL ;	//INC10
   A_INC100 : BOOL ;	//INC100
   A_INC1000 : BOOL ;	//INC1000
   A_INC10000 : BOOL ;	//INC10000
   A_INCVar : BOOL ;	//INC variable
   A_OEMAxis : BYTE ;	//OEM axis signals
   A_InvHWDirOfRot : BOOL ;	// Inverting handwheel direction of rotation
   f7_1 : BOOL ;
   f7_2 : BOOL ;
   f7_3 : BOOL ;
   f7_4 : BOOL ;
   f7_5 : BOOL ;
   f7_6 : BOOL ;
   f7_7 : BOOL ;
   A_NCASpChanA : BOOL ;	//Assign NC axis/spindle channel A
   A_NCASpChanB : BOOL ;	//Assign NC axis/spindle channel B
   A_NCASpChanC : BOOL ;	//Assign NC axis/spindle channel C
   A_NCASpChanD : BOOL ;	//Assign NC axis/spindle channel D
   A_NCASpStrobe : BOOL ;	//Activation of assignment with pos. edge
   f8_5 : BOOL ;
   f8_6 : BOOL ;
   A_PLCASp : BOOL ;	//Request PLC axis/spindle
   A_Para_A : BOOL ;	//Parameter block servo A
   A_Para_B : BOOL ;	//Parameter block servo B
   A_Para_C : BOOL ;	//Parameter block servo C
   A_LockParSetDef : BOOL ;	//Lock parameter set definition from NC
   f9_4 : BOOL ;
   f9_5 : BOOL ;
   f9_6 : BOOL ;
   f9_7 : BOOL ;
   A_REPOSDelay : BOOL ;	//REPOS DELAY
   f10_1 : BOOL ;
   f10_2 : BOOL ;
   f10_3 : BOOL ;
   f10_4 : BOOL ;
   f10_5 : BOOL ;
   f10_6 : BOOL ;
   f10_7 : BOOL ;
   A_StartBrakeTest : BOOL ;	// Start brake test
   f11_1 : BOOL ;
   f11_2 : BOOL ;
   f11_3 : BOOL ;
   f11_4 : BOOL ;
   f11_5 : BOOL ;
   f11_6 : BOOL ;
   f11_7 : BOOL ;
   A_HWLimitMinus : BOOL ;	//Hardware limit switch minus
   A_HWLimitPlus : BOOL ;	//Hardware limit switch plus
   A_SWLimit2Minus : BOOL ;	//2nd software limit switch minus
   A_SWLimit2Plus : BOOL ;	//2nd software limit switch plus
   A_ModuloLimitEn : BOOL ;	// Modulo limit enabled
   f12_5 : BOOL ;
   f12_6 : BOOL ;
   A_DelayRef : BOOL ;	//Delay reference point approach
   A_JogFixPPos0 : BOOL ;	// JogFixPointPos 0
   A_JogFixPPos1 : BOOL ;	// JogFixPointPos 1
   A_JogFixPPos2 : BOOL ;	// JogFixPointPos 2
   A_JogToPos : BOOL ;	// Jog to position
   f13_4 : BOOL ;
   f13_5 : BOOL ;
   f13_6 : BOOL ;
   f13_7 : BOOL ;
   A_ProgtestSuppress : BOOL ;	// Program test to supress
   A_ProgtestActivate : BOOL ;	// Program test activate
   f14_2 : BOOL ;
   f14_3 : BOOL ;
   f14_4 : BOOL ;
   f14_5 : BOOL ;
   f14_6 : BOOL ;
   f14_7 : BOOL ;
   f15 : BYTE ;
   A_ActGearA : BOOL ;	//Actual gear stage A
   A_ActGearB : BOOL ;	//Actual gear stage B
   A_ActGearC : BOOL ;	//Actual gear stage C
   A_GearChangeOv : BOOL ;	//Gear has changed over
   A_Sp1Syn : BOOL ;	//Re-synchronize spindle 1
   A_Sp2Syn : BOOL ;	//Re-synchronize spindle 2
   A_NoMonitorGear : BOOL ;	//No monitoring when changing gear
   A_DeleteS : BOOL ;	//Delete S value
   A_FD_ORSp : BOOL ;	//Feedrate override for spindle valid
   f17_1 : BOOL ;
   f17_2 : BOOL ;
   f17_3 : BOOL ;
   A_Sp1SynP : BOOL ;	//Re-synchronize spindle 1 f. positioning
   A_Sp2SynP : BOOL ;	//Re-synchronize spindle 2 f. positioning
   A_M3M4Inv : BOOL ;	//Invert M3/M4
   f17_7 : BOOL ;
   f18_0 : BOOL ;
   f18_1 : BOOL ;
   f18_2 : BOOL ;
   f18_3 : BOOL ;
   A_OscilPLC : BOOL ;	//Oscillation via PLC
   A_OscilSpeed : BOOL ;	//enable Oscillation
   A_SetRotDirectRight : BOOL ;	//Setpoint osci. direct. right
   A_SetRotDirectLeft : BOOL ;	//Setpoint osci. direct. left
   A_SpOR : BYTE ;	//Spindle override
   f20_0 : BOOL ;
   A_RUEncQuStop : BOOL ;	//Run-up encoder quick stop
   f20_2 : BOOL ;
   A_SpeedSetpSmooth : BOOL ;	//Speed setpoint smoothing
   f20_4 : BOOL ;
   A_HoldBrakeToOpen : BOOL ;	// holding brake open
   f20_6 : BOOL ;
   f20_7 : BOOL ;
   A_ParA : BOOL ;	//Parameter set selection A
   A_ParB : BOOL ;	//Parameter set selection B
   A_ParC : BOOL ;	//Parameter set selection C
   A_MotA : BOOL ;	//Motor selection A
   A_MotB : BOOL ;	//Motor selection B
   A_MotOK : BOOL ;	//Motor selected
   A_IntegratDisable : BOOL ;	//n controller integrator disable
   A_PulseEnable : BOOL ;	//Pulse enable
   A_SG_SBH : BOOL ;	//Deselection SG/SBH
   A_SBH : BOOL ;	//Deselection of safe standstill
   f22_2 : BOOL ;
   A_SGselect0 : BOOL ;	//Selection SG bit 0
   A_SGselect1 : BOOL ;	//Selection SG bit 1
   f22_5 : BOOL ;
   f22_6 : BOOL ;
   f22_7 : BOOL ;
   A_Transmiss0 : BOOL ;	//Selection Transmission bit 0
   A_Transmiss1 : BOOL ;	//Selection Transmission bit 1
   A_Transmiss2 : BOOL ;	//Selection Transmission bit 2
   f23_3 : BOOL ;
   A_SE : BOOL ;	//Selection SE
   A_BrakeToClose : BOOL ;	//Sinamics: Brake to close
   f23_6 : BOOL ;
   A_TestStop : BOOL ;	//Activate test stop
   A_RotationMonit : BOOL ;	// Stepper motor: Rotation monitoring
   A_ControlAx : BOOL ;	// Control Axis
   f24_2 : BOOL ;
   f24_3 : BOOL ;
   A_TorqComp : BOOL ;	// Torque compensation
   A_ChangSetpOutAss0 : BOOL ;	// Bit value for CTRLOUT_changed - Change setpoint output assignment
   A_ChangSetpOutAss1 : BOOL ;	// Bit value for CTRLOUT_changed - Change setpoint output assignment
   A_MS : BOOL ;	//Master / Slave On
   f25 : BYTE ;
   f26_0 : BOOL ;
   f26_1 : BOOL ;
   f26_2 : BOOL ;
   A_CompContr : BOOL ;	//Compensation controller On
   A_FollowAxOv : BOOL ;	//Enable following axis override
   f26_5 : BOOL ;
   f26_6 : BOOL ;
   f26_7 : BOOL ;
   A_DEPMCS : BOOL ;	// Resume: DEPMCS
   A_DEPBCS : BOOL ;	// Resume: DEPBCS
   A_Corr : BOOL ;	// Resume: Corr
   A_HIAxMove : BOOL ;	// Resume: HIAxMove
   A_StopDEPMCS : BOOL ;	// Stop: DEPMCS
   A_StopDEPBCS : BOOL ;	// Stop: DEPBCS
   A_StopCorr : BOOL ;	// Stop: Corr
   A_StopHIAxMove : BOOL ;	// Stop: HIAxMove
   A_OscillAxExtRev : BOOL ;	// OscillAxExtReversal
   A_AxReset : BOOL ;	// AXRESET
   A_AxResume : BOOL ;	// AXRESUME
   A_SetRP : BOOL ;	//Set reversal point
   A_ChangeRP : BOOL ;	//Change reversal point
   A_StopRP : BOOL ;	//Stop at next reversal point
   A_Stop : BOOL ;	//Stop
   A_PLCAxis : BOOL ;	//PLC checks axis
   f29_0 : BOOL ;
   f29_1 : BOOL ;
   f29_2 : BOOL ;
   f29_3 : BOOL ;
   A_StartGantSynRun : BOOL ;	//Start gantry synchronization run
   A_NoAutoSync : BOOL ;	//No auto sync
   f29_6 : BOOL ;
   f29_7 : BOOL ;
   A_StopSpindle : BOOL ;	//Stop spindle
   A_StartCW : BOOL ;	//Start spindle Clockwise
   A_StartCCW : BOOL ;	//Start spindle Counterclockwise
   A_AutoGearStep : BOOL ;	//Autom. gear step change
   A_PosSpindle : BOOL ;	//Position spindle
   f30_5 : BOOL ;
   f30_6 : BOOL ;
   f30_7 : BOOL ;
   f31_0 : BOOL ;
   f31_1 : BOOL ;
   f31_2 : BOOL ;
   f31_3 : BOOL ;
   A_Resynchronize : BOOL ;	// Resynchronize
   A_DisSync : BOOL ;	// Disable synchronization
   A_Tracksync : BOOL ;	// Track synchronism
   A_DelSyncRunCorr : BOOL ;	// Deleting synchronous run correction
   f32_0 : BOOL ;
   f32_1 : BOOL ;
   A_extStopA : BOOL ;	//Deselection external Stop A
   A_extStopC : BOOL ;	//Deselection external Stop C
   A_extStopD : BOOL ;	//Deselection external Stop D
   A_extStopE : BOOL ;	//Deselection external Stop E
   f32_6 : BOOL ;
   f32_7 : BOOL ;
   f33_0 : BOOL ;
   f33_1 : BOOL ;
   f33_2 : BOOL ;
   f33_3 : BOOL ;
   A_SGcorr_0 : BOOL ;	//Selection SG-correction Bit 0
   A_SGcorr_1 : BOOL ;	//Selection SG-correction Bit 1
   A_SGcorr_2 : BOOL ;	//Selection SG-correction Bit 2
   A_SGcorr_3 : BOOL ;	//Selection SG-correction Bit 3
   f34 : ARRAY  [34 .. 55 ] OF BYTE ;
   A_FeedDriveCAxEng : BOOL ;	// Seperate feed drive as C axis engaged
   A_SpSpeedDisp : BOOL ;	// Spindle speed display
   A_SpInsideClamp : BOOL ;	// Spindle inside clamping
   f56_3 : BOOL ;
   f56_4 : BOOL ;
   f56_5 : BOOL ;
   f56_6 : BOOL ;
   f56_7 : BOOL ;
   f57 : BYTE ;
   f58 : WORD ;	// FC18: internal
   E_SpNA : BOOL ;	//Spindle/no axis
   E_NCU_Link : BOOL ;	//NCU_link active axis
   E_EncodFreq1 : BOOL ;	//Encoder limit frequency 1 exceeded
   E_EncodFreq2 : BOOL ;	//Encoder limit frequency 2 exceeded
   E_RefSyn1 : BOOL ;	//Referenced/synchronized 1
   E_RefSyn2 : BOOL ;	//Referenced/synchronized 2
   E_ExactCoarse : BOOL ;	//Position reached with exact stop coarse
   E_ExactFine : BOOL ;	//Position reached with exact stop fine
   E_TravRequ : BOOL ;	//Travel request
   E_AxialAlarm : BOOL ;	// Axial alarm
   E_AxisReady : BOOL ;	//Axis ready
   E_Follow_upMode : BOOL ;	//Follow-up mode active
   E_Stat : BOOL ;	//Axis/spindle stationary (n<nmin)
   E_PositContr : BOOL ;	//Position controller active
   E_SpeedContr : BOOL ;	//Speed controller active
   E_CurrentContr : BOOL ;	//Current controller active
   E_SWCam : BOOL ;	//Software cams active
   E_HWOverlay : BOOL ;	//Handwheel overlay active
   E_RevFD : BOOL ;	//Revolutional feedrate active
   E_MeasAct : BOOL ;	//Measuring active
   E_ActTravFStop : BOOL ;	//Activate travel to fixed stop
   E_FixedStop : BOOL ;	//Fixed stop reached
   E_ForceFixedStop : BOOL ;	// Force fixed stop limited
   E_AxContainerRot : BOOL ;	// Axis container rotation active
   E_AxReset : BOOL ;	// Axis reset done
   E_PLCCtrlAx : BOOL ;	// PLCcontrolled axis
   E_AxStop : BOOL ;	// Axis stop active
   E_AxSpDisable : BOOL ;	// Axis/spindle disable active
   E_StopDEPMCS : BOOL ;	// stop DEPMCS active
   E_StopDEPBCS : BOOL ;	// stop DEPBCS active
   E_StopCorr : BOOL ;	// stop Corr active
   E_StopHIAxMove : BOOL ;	// Stop HIAxMove active
   E_HW1 : BOOL ;	//Handwheel 1 active
   E_HW2 : BOOL ;	//Handwheel 2 active
   E_HW3 : BOOL ;	//Handwheel 3 active
   f64_3 : BOOL ;
   E_TReqMinus : BOOL ;	// Travel request minus
   E_TReqPlus : BOOL ;	// Travel request plus
   E_TCMinus : BOOL ;	//Traverse command minus
   E_TCPlus : BOOL ;	//Traverse command plus
   E_INC1 : BOOL ;	//INC1
   E_INC10 : BOOL ;	//INC10
   E_INC100 : BOOL ;	//INC100
   E_INC1000 : BOOL ;	//INC1000
   E_INC10000 : BOOL ;	//INC10000
   E_INCVar : BOOL ;	//INC variable
   f65_6 : BOOL ;
   f65_7 : BOOL ;
   E_OEMAxis : BYTE ;	//OEM axis signals
   E_InvHWDirOfRot : BOOL ;	// Handwheel direction of rotation invert actively
   f67_1 : BOOL ;
   f67_2 : BOOL ;
   f67_3 : BOOL ;
   f67_4 : BOOL ;
   f67_5 : BOOL ;
   f67_6 : BOOL ;
   f67_7 : BOOL ;
   E_NCASpChanA : BOOL ;	//NC axis/spindle in channel A
   E_NCASpChanB : BOOL ;	//NC axis/spindle in channel B
   E_NCASpChanC : BOOL ;	//NC axis/spindle in channel C
   E_NCASpChanD : BOOL ;	//NC axis/spindle in channel D
   E_PLCType : BOOL ;	//New type requested by PLC
   E_ChPoss : BOOL ;	//Change axis possible
   E_NeutrASp : BOOL ;	//Neutral axis/spindle
   E_PLCASp : BOOL ;	//PLC axis/spindle
   E_ParS_A : BOOL ;	//Parameter block servo A
   E_ParS_B : BOOL ;	//Parameter block servo B
   E_ParS_C : BOOL ;	//Parameter block servo C
   E_NCUNumLink_3 : BOOL ;
   E_NCUNumLink_4 : BOOL ;
   E_NCUNumLink_5 : BOOL ;
   E_NCUNumLink_6 : BOOL ;
   E_NCUNumLink_7 : BOOL ;
   E_ReposSh : BOOL ;	// Repos shift
   E_ReposShValid : BOOL ;	// Repos shift valid
   E_ReposDelayQuit : BOOL ;	// Repos delay quit
   f70_3 : BOOL ;
   f70_4 : BOOL ;
   f70_5 : BOOL ;
   f70_6 : BOOL ;
   f70_7 : BOOL ;
   E_BrakeTest : BOOL ;	// Brake test active
   f71_1 : BOOL ;
   f71_2 : BOOL ;
   f71_3 : BOOL ;
   E_POS_RESTORED1 : BOOL ;	// POS_RESTORED 1
   E_POS_RESTORED2 : BOOL ;	// POS_RESTORED 2
   f71_6 : BOOL ;
   E_PLCAxDedic : BOOL ;	// PLC Axis dedicated
   E_MMC_REPOSDelay : BOOL ;	//MMC REPOS DELAY
   f72_1 : BOOL ;
   f72_2 : BOOL ;
   f72_3 : BOOL ;
   f72_4 : BOOL ;
   f72_5 : BOOL ;
   f72_6 : BOOL ;
   f72_7 : BOOL ;
   f73 : BYTE ;
   f74_0 : BOOL ;
   f74_1 : BOOL ;
   f74_2 : BOOL ;
   f74_3 : BOOL ;
   E_ModLimEnAct : BOOL ;	// Modulo limit enabled active
   f74_5 : BOOL ;
   f74_6 : BOOL ;
   f74_7 : BOOL ;
   E_JogFixPPos0Act : BOOL ;	// JogFixPointPos 0 active
   E_JogFixPPos1Act : BOOL ;	// JogFixPointPos 1 active
   E_JogFixPPos2Act : BOOL ;	// JogFixPointPos 2 active
   E_JogFixPPos0 : BOOL ;	// JogFixPointPos 0 reached
   E_JogFixPPos1 : BOOL ;	// JogFixPointPos 1 reached
   E_JogFixPPos2 : BOOL ;	// JogFixPointPos 2 reached
   E_JogToPos : BOOL ;	// Jog to position active
   E_JogPos : BOOL ;	// Jog position reached
   E_ScratchPulse : BOOL ;	//Scratch pulse
   f76_1 : BOOL ;
   f76_2 : BOOL ;
   f76_3 : BOOL ;
   E_PathAxis : BOOL ;	// Path axis
   E_PosAxis : BOOL ;	//Positioning axis
   E_IndexAxisPos : BOOL ;	//Indexing axis in position
   E_CurvePos : BOOL ;	//Curve axis in position
   E_CollCheckRedSpeed : BOOL ;	//reduced speed of Collisions Check
   f77_1 : BOOL ;
   f77_2 : BOOL ;
   f77_3 : BOOL ;
   f77_4 : BOOL ;
   f77_5 : BOOL ;
   f77_6 : BOOL ;
   f77_7 : BOOL ;
   E_FPosAxis : REAL ;	//F function (REAL format) for positioning axes
   E_SetpGearA : BOOL ;	//Setpoint gear stage A
   E_SetpGearB : BOOL ;	//Setpoint gear stage B
   E_SetpGearC : BOOL ;	//Setpoint gear stage C
   E_GearChange : BOOL ;	//Gear changeover
   f82_4 : BOOL ;
   f82_5 : BOOL ;
   f82_6 : BOOL ;
   f82_7 : BOOL ;
   E_SpeedLimit : BOOL ;	//Speed limit exceeded
   E_SetSpeedLimit : BOOL ;	//Setpoint speed limited
   E_SetSpeedIncreased : BOOL ;	//Setpoint speed increased
   E_GeoMonit : BOOL ;	//Geometry monitoring
   E_SupportAreaViol : BOOL ;	//Support area limits violated
   E_SetRange : BOOL ;	//Spindle in setpoint range
   E_SpeedMonit : BOOL ;	//Speed monitoring
   E_ActRotRight : BOOL ;	//Actual rotation direction right
   E_ConstCuttSpeed : BOOL ;	//Const. cutting speed active
   E_SUG : BOOL ;	//SUG active (grinding wheel surface speed)
   E_CLG : BOOL ;	//CLG active
   E_Tapping : BOOL ;	//Tapping without compensating chuck
   E_SyncMode : BOOL ;	//Synchronous mode spindle active
   E_PosMode : BOOL ;	//Positioning mode spindle active
   E_OscillMode : BOOL ;	//Oscillation mode spindle active
   E_ContrMode : BOOL ;	//Control mode spindle active
   E_ToolDynLimit : BOOL ;	// Tool with limit of dynamics
   f85_1 : BOOL ;
   f85_2 : BOOL ;
   f85_3 : BOOL ;
   f85_4 : BOOL ;
   E_SpInPosition : BOOL ;	// Spindle in position
   f85_6 : BOOL ;
   f85_7 : BOOL ;
   E_MFunct : INT ;	//M function (INT) for spindle
   E_SFunct : REAL ;	//S function (REAL) for spindle
   f92_0 : BOOL ;
   E_RUEncDisabl : BOOL ;	//Run-up encoder disable active
   f92_2 : BOOL ;
   E_SpeedSetpSmooth : BOOL ;	//Speed setpoint smoothing active
   E_RLIact : BOOL ;	// RLI active
   E_HoldBrakeOpened : BOOL ;	// Holding brake opened
   f92_6 : BOOL ;
   f92_7 : BOOL ;
   E_ParA : BOOL ;	//Active parameter set A
   E_ParB : BOOL ;	//Active parameter set B
   E_ParC : BOOL ;	//Active parameter set C
   E_MotA : BOOL ;	//Active motor A
   E_MotB : BOOL ;	//Active motor B
   E_MotOK : BOOL ;	//Drive ready
   E_IntegratDisable : BOOL ;	//n controller integrator disabled
   E_PulseEnable : BOOL ;	//Pulses enabled
   E_MTempWarn : BOOL ;	//Temperature prewarning motor
   E_HTempWarn : BOOL ;	//Temperature prewarning heat sink
   E_RUComplete : BOOL ;	//Ramp-up complete
   E_MdMdx : BOOL ;	//Md<Mdx
   E_NactNmin : BOOL ;	//nact<nmin
   E_NactNx : BOOL ;	//nact<nx
   E_NactNset : BOOL ;	//nact<nset
   E_Message : BOOL ;	//Variable message function
   E_UDClessAlThreshold : BOOL ;	//UDC-link < alarm threshold
   f95_1 : BOOL ;
   f95_2 : BOOL ;
   f95_3 : BOOL ;
   f95_4 : BOOL ;
   f95_5 : BOOL ;
   f95_6 : BOOL ;
   f95_7 : BOOL ;	// Power Section I2T limit
   E_SpindleMonit : BOOL ;	//Error spindle monitoring
   E_AxisCtrl : BOOL ;	// Axis control active
   E_MSFine : BOOL ;	// Master/Slave fine
   E_MSCoarse : BOOL ;	// Master/Slave coarse
   E_MSCompContr : BOOL ;	// Master/Slave Compensation controller activ
   E_BitValCtrlOutChang0 : BOOL ;	// Bit value for CTRLOUT_changed 0:  Change setpoint output assignment
   E_BitValCtrlOutChang1 : BOOL ;	// Bit value for CTRLOUT_changed 1:  Change setpoint output assignment
   E_MS : BOOL ;	//Master/ slave active
   f97 : BYTE ;
   E_SyncronFine : BOOL ;	//Synchronism fine
   E_SyncronCoarse : BOOL ;	//Synchronism coarse
   E_ActValCoupling : BOOL ;	//Actual value coupling
   f98_3 : BOOL ;
   E_OverlayMotion : BOOL ;	//Overlaid motion
   E_SWL : BOOL ;	//Speed warning limit reached
   E_AWL : BOOL ;	//Acceleration warning limit reached
   E_EmRetr : BOOL ;	//Emergency retraction active
   E_MasterSp : BOOL ;	//Master spindle
   E_SlaveSp : BOOL ;	//Slave spindle
   E_SyncRunCorrDOut : BOOL ;	// Synchronous run correction driven out
   E_AxisAccel : BOOL ;	//Axis accelerated
   E_Sync : BOOL ;	//Synchronization active
   E_MSR : BOOL ;	//Max speed reached
   E_MAR : BOOL ;	//Max acceleration reached
   f99_7 : BOOL ;
   f100_0 : BOOL ;
   f100_1 : BOOL ;
   E_OscillAxExtRev : BOOL ;	// OscillAxExt Reversal active
   E_StopOscill : BOOL ;	//Oscillation cannot start
   E_ErrorOscill : BOOL ;	//Error during oscillation
   E_SparkOut : BOOL ;	//Spark-out active
   E_OscillMotion : BOOL ;	//Oscillation motion active
   E_Oscill : BOOL ;	//Oscillation active
   f101_0 : BOOL ;
   f101_1 : BOOL ;
   E_GantCOLimit : BOOL ;	//Gantry cut-off limit exceeded
   E_GantWarn : BOOL ;	//Gantry warning limit exceeded
   E_SynRunStart : BOOL ;	//Synchronization run ready to start
   E_GantGroupSyn : BOOL ;	//Gantry grouping is synchronous
   E_GantLeadAxis : BOOL ;	//Gantry leading axis
   E_GantAxis : BOOL ;	//Gantry axis
   f102 : BYTE ;
   E_SyncRunCorrIncl : BOOL ;	// Synchronous run correction is included
   f103_1 : BOOL ;
   f103_2 : BOOL ;
   f103_3 : BOOL ;
   f103_4 : BOOL ;
   f103_5 : BOOL ;
   f103_6 : BOOL ;
   f103_7 : BOOL ;
   E_AIAxis : ARRAY  [1 .. 31 ] OF BOOL ;	//Active infeed axis[1..31]
   E_SG_SBH : BOOL ;	//Active SG/SBH
   E_ErrLifeS_CRC : BOOL ;	// Error lifesign or CRC-error
   E_ImpdelNCK : BOOL ;	//Delete pulses NCK
   r108_3 : BOOL ;
   r108_4 : BOOL ;
   r108_5 : BOOL ;
   r108_6 : BOOL ;
   E_SRef : BOOL ;	//Axis safely referenced
   E_SN1Plus : BOOL ;	//Actual position > cam position SN1+
   E_SN1Minus : BOOL ;	//Actual position > cam position SN1-
   E_SN2Plus : BOOL ;	//Actual position > cam position SN2+
   E_SN2Minus : BOOL ;	//Actual position > cam position SN2-
   E_SN3Plus : BOOL ;	//Actual position > cam position SN3+
   E_SN3Minus : BOOL ;	//Actual position > cam position SN3-
   E_SN4Plus : BOOL ;	//Actual position > cam position SN4+
   E_SN4Minus : BOOL ;	//Actual position > cam position SN4-
   f110_0 : BOOL ;
   E_SBH : BOOL ;	//Active SBH
   f110_2 : BOOL ;
   E_SG_0 : BOOL ;	//Active SG 0
   E_SG_1 : BOOL ;	//Active SG 1
   E_n_nx : BOOL ;	//n < nx
   f110_6 : BOOL ;
   f110_7 : BOOL ;
   f111_0 : BOOL ;
   f111_1 : BOOL ;
   f111_2 : BOOL ;
   f111_3 : BOOL ;
   E_StopAB : BOOL ;	//Stop A/B active
   E_StopC : BOOL ;	//Stop C active
   E_StopD : BOOL ;	//Stop D active
   E_StopE : BOOL ;	//Stop E active
   E_CamRangeTr1 : BYTE ;	//Cam Range for Cam Track 1
   E_CamRangeTr2 : BYTE ;	//Cam Range for Cam Track 2
   E_CamRangeTr3 : BYTE ;	//Cam Range for Cam Track 3
   E_CamRangeTr4 : BYTE ;	//Cam Range for Cam Track 4
   f116 : BYTE ;
   E_CamTrack1 : BOOL ;	//Cam Track 1
   E_CamTrack2 : BOOL ;	//Cam Track 2
   E_CamTrack3 : BOOL ;	//Cam Track 3
   E_CamTrack4 : BOOL ;	//Cam Track 4
   f117_4 : BOOL ;
   f117_5 : BOOL ;
   f117_6 : BOOL ;
   f117_7 : BOOL ;
   E_CamRangeBitTr1 : ARRAY  [0 .. 14 ] OF //Cam Range Bits for Cam Track 1
   BOOL ;
   E_CamRangeBitTr2 : ARRAY  [0 .. 14 ] OF //Cam Range Bits for Cam Track 2
   BOOL ;
   E_CamRangeBitTr3 : ARRAY  [0 .. 14 ] OF //Cam Range Bits for Cam Track 3
   BOOL ;
   E_CamRangeBitTr4 : ARRAY  [0 .. 14 ] OF //Cam Range Bits for Cam Track 4
   BOOL ;
   f126 : WORD ;	// internal
   E_MMC_ProgtestSuppress : BOOL ;	// HMI->PLC: Program test to supress
   E_MMC_ProgtestActivate : BOOL ;	// HMI->PLC: Program test activate
   f128_2 : BOOL ;
   f128_3 : BOOL ;
   f128_4 : BOOL ;
   f128_5 : BOOL ;
   f128_6 : BOOL ;
   f128_7 : BOOL ;
   f129 : BYTE ;
   f130 : WORD ;
   E_SensorAv : BOOL ;	// Sensors available
   E_S1aMeasARod : BOOL ;	// Sensor S1: analogous measurement position of actuating rod
   f132_2 : BOOL ;
   f132_3 : BOOL ;
   E_S4dPistonStopP : BOOL ;	// Sensor S4: digital value piston stop position
   E_S5dAngleShaft : BOOL ;	// Sensor S5: digital value angle situation shaft
   f132_6 : BOOL ;
   f132_7 : BOOL ;
   f133 : BYTE ;
   E_ClampingState : INT ;	// state of the clamping system
   E_AnalogSensor : INT ;	// analog sensor on the motor
   f138_0 : BOOL ;
   f138_1 : BOOL ;
   f138_2 : BOOL ;
   f138_3 : BOOL ;
   E_S4PistonStopP : BOOL ;	// Sensor S4: piston stop position
   E_S5AngleShaft : BOOL ;	// Sensor S5: angle situation shaft
   f138_6 : BOOL ;
   f138_7 : BOOL ;
   f139 : BYTE ;
  END_STRUCT ;	
END_TYPE

TYPE UDT 71
VERSION : 0.0
  STRUCT
   IFNo : ARRAY  [1 .. 16 ] OF BOOL ;	//Interface [no.] active
   Quit : ARRAY  [1 .. 16 ] OF BOOL ;	//perform Quit-End
   IF : ARRAY  [1 .. 16 ] OF STRUCT
    Loading : BOOL ;
    Unloading : BOOL ;
    Reloading : BOOL ;
    Positioning : BOOL ;
    PosbyProgram : BOOL ;	//Initiation by CNC Program
    PositioningMT : BOOL ;	//Positioning Multitool
    f0_6 : BOOL ;
    f0_7 : BOOL ;
    PerfStatusError : BOOL ;
    n1_1 : BOOL ;
    n1_2 : BOOL ;
    n1_3 : BOOL ;
    n1_4 : BOOL ;
    n1_5 : BOOL ;
    n1_6 : BOOL ;
    DataInDB1071 : BOOL ;
    Channel : BYTE ;	//Assigned channel
    TMno : BYTE ;	//Tool management no.
    Free1 : DINT ;	//Unassigned parameter 1
    Free2 : DINT ;	//Unassigned parameter 2
    Free3 : DINT ;	//Unassigned parameter 3
    IdentLoad : INT ;	//Identification for loading/unloading station
    NoLoad : INT ;	//No. of loading station
    SMag : INT ;	//Magazine no. (source) for unloading/reloading/pos.
    SLoc : INT ;	//Location no. (source) for unloading/reloading/pos.
    TMag : INT ;	//Magazine no. (target) for loading/reloading
    TLoc : INT ;	//Location no. (target) for loading/reloading
    WithoutMagMoving : BOOL ;	//HMI Data: Without Magazine Moving
    Res2 : BYTE ;
   END_STRUCT ;
  END_STRUCT ;	
END_TYPE

TYPE UDT 72
VERSION : 0.0
  STRUCT
   IFNo : ARRAY  [1 .. 16 ] OF BOOL ;	//Interface [no.] active
   Quit : ARRAY  [1 .. 16 ] OF BOOL ;	//perform Quit-End
   IF : ARRAY  [1 .. 16 ] OF STRUCT
    Comp : BOOL ;	//Compulsory change
    Perform : BOOL ;	//Perform change
    Prepare : BOOL ;	//Prepare change
    T0 : BOOL ;	//T0 programmed
    OldTinDBW42 : BOOL ;	//ZWS No. of Old Tool in DBW (n+42)
    ManTIn : BOOL ;	//Put in Tool in Spindle manual
    ManTOut : BOOL ;	//Get out Tool from Spindle manual
    SpiTRSpi : BOOL ;	//Spindle Tool remains in spindle
    PerfStatusError : BOOL ;
    n1_1 : BOOL ;
    n1_2 : BOOL ;
    n1_3 : BOOL ;
    n1_4 : BOOL ;
    n1_5 : BOOL ;
    n1_6 : BOOL ;
    DataInDB1072 : BOOL ;
    Channel : BYTE ;	//Assigned channel
    TMno : BYTE ;	//Tool management no.
    Free1 : DINT ;	//Unassigned parameter 1
    Free2 : DINT ;	//Unassigned parameter 2
    Free3 : DINT ;	//Unassigned parameter 3
    IdentBuff : INT ;	//Buffer identification (fixed value 9998)
    NoBuff : INT ;	//Relative location (target) in the buffer
    SMag : INT ;	//Magazine no. (source) for new tool
    SLoc : INT ;	//Location no. (source) for new tool
    TMag : INT ;	//Magazine no. (target) for old tool
    TLoc : INT ;	//Location no. (target) for old tool
    LocType : INT ;	//Tool new: location type
    SLeft : INT ;	//Tool new: size left
    SRight : INT ;	//Tool new: size right
    STop : INT ;	//Tool new: size top
    SBottom : INT ;	//Tool new: size bottom
    ToolInBuff : BOOL ;	//ID for tools in buffer
    IgnoreDisab : BOOL ;	//Ignore disabled
    TBUnloaded : BOOL ;	//To be unloaded
    TBLoaded : BOOL ;	//To be loaded
    MasterTool : BOOL ;	//Master tool
    n38_5 : BOOL ;	//reserved
    Exchange_1to1 : BOOL ;	//1:1 exchange
    HandTool : BOOL ;	//Hand tool
    ActTool : BOOL ;	//Active tool
    ToolEnabl : BOOL ;	//Tool enabled
    ToolDisab : BOOL ;	//Tool disabled
    Measured : BOOL ;	//Tool measured
    Prewarn : BOOL ;	//Prewarning limit reached
    ToolChange : BOOL ;	//Tool being changed
    FixedLoc : BOOL ;	//Tool fixed location coded
    ToolUsed : BOOL ;	//Tool was in use
    T_no : INT ;	//Tool new: T no.
    OldTZWSNo : INT ;	//ZWS No. of Old Tool
    MyMag : INT ;
    MyPlace : INT ;
   END_STRUCT ;
  END_STRUCT ;	
END_TYPE

TYPE UDT 73
VERSION : 0.0
  STRUCT
   IfNo : ARRAY  [1 .. 16 ] OF BOOL ;	//Interface [no.] active
   Quit : ARRAY  [1 .. 16 ] OF BOOL ;	//perform Quit-End
   IF : ARRAY  [1 .. 16 ] OF STRUCT
    Comp : BOOL ;	//Compulsory change
    Perform : BOOL ;	//Perform change
    f0_2 : BOOL ;
    T0 : BOOL ;	//T0 programmed
    f0_4 : BOOL ;
    f0_5 : BOOL ;
    ManTOut : BOOL ;	//Get out Tool from Holder manual
    f0_7 : BOOL ;
    PerfStatusError : BOOL ;
    n1_1 : BOOL ;
    n1_2 : BOOL ;
    n1_3 : BOOL ;
    n1_4 : BOOL ;
    n1_5 : BOOL ;
    n1_6 : BOOL ;
    DataInDB1073 : BOOL ;
    Channel : BYTE ;	//Assigned channel
    TMno : BYTE ;	//Tool management no.
    Free1 : DINT ;	//Unassigned parameter 1
    Free2 : DINT ;	//Unassigned parameter 2
    Free3 : DINT ;	//Unassigned parameter 3
    KennZWS : INT ;	//Reserved (buffer identification)
    NoBuff : INT ;	//Rel. location in buffer (res.)
    SMag : INT ;	//Magazine no. of turret
    SLoc : INT ;	//Location no. for new tool
    TMag : INT ;	//Magazine no. of turret (res.)
    TLoc : INT ;	//Location no. for old tool
    LocType : INT ;	//Tool new: location type
    SLeft : INT ;	//Tool new: size left
    SRight : INT ;	//Tool new: size right
    STop : INT ;	//Tool new: size top
    SBottom : INT ;	//Tool new: size bottom
    ToolInBuff : BOOL ;	//ID for tools in buffer
    IgnoreDisab : BOOL ;	//Ignore disabled
    TBUnloaded : BOOL ;	//To be unloaded
    TBLoaded : BOOL ;	//To be loaded
    MasterTool : BOOL ;	//Master tool
    n38_5 : BOOL ;	//reserved
    Exchange_1to1 : BOOL ;	//1:1 exchange
    HandTool : BOOL ;	//Hand tool
    ActTool : BOOL ;	//Active tool
    ToolEnabl : BOOL ;	//Tool enabled
    ToolDisab : BOOL ;	//Tool disabled
    Measured : BOOL ;	//Tool measured
    Prewarn : BOOL ;	//Prewarning limit reached
    ToolChange : BOOL ;	//Tool being changed
    FixedLoc : BOOL ;	//Tool fixed location coded
    ToolUsed : BOOL ;	//Tool was in use
    T_no : INT ;	//Tool new: T no.
    MyPlace : INT ;
   END_STRUCT ;
  END_STRUCT ;	
END_TYPE

TYPE UDT 77
VERSION : 0.0
  STRUCT
   MCP1In : ARRAY  [0 .. 7 ] OF BYTE ;
   MCP1Out : ARRAY  [0 .. 7 ] OF BYTE ;
   MCP1StatSend : DWORD ;
   MCP1StatRec : DWORD ;
   MCP2In : ARRAY  [0 .. 7 ] OF BYTE ;
   MCP2Out : ARRAY  [0 .. 7 ] OF BYTE ;
   MCP2StatSend : DWORD ;
   MCP2StatRec : DWORD ;
   BHGIn : ARRAY  [0 .. 5 ] OF BYTE ;
   Filler : ARRAY  [0 .. 5 ] OF BYTE ;
   BHGOut : ARRAY  [0 .. 19 ] OF BYTE ;
   BHGStatSend : DWORD ;
   BHGStatRec : DWORD ;
  END_STRUCT ;	
END_TYPE

TYPE UDT 1002
VERSION : 0.0
  STRUCT 	//Offset 0
   Chan : ARRAY  [1 .. 10 ] OF STRUCT 	//From Channel 1 to Channel 10
    FDD : ARRAY  [0 .. 15 ] OF //Feed disable
    BOOL ;
    RID : ARRAY  [0 .. 15 ] OF //Read-in disable
    BOOL ;
    NCSD : ARRAY  [0 .. 15 ] OF //NC start disable
    BOOL ;
    FdStop_1 : ARRAY  [0 .. 15 ] OF //Feed stop GEOaxis 1
    BOOL ;
    FdStop_2 : ARRAY  [0 .. 15 ] OF //Feed stop GEOaxis 2
    BOOL ;
    FdStop_3 : ARRAY  [0 .. 15 ] OF //Feed stop GEOaxis 3
    BOOL ;
   END_STRUCT ;	//without Alarmno for Chan (120 Byte)
//Offset 120
   Axis : ARRAY  [1 .. 31 ] OF STRUCT 	//From Axis 1 to Axis 31
    FdStop : ARRAY  [0 .. 15 ] OF //Feed stop axis/spindle 1
    BOOL ;
   END_STRUCT ;	//without Alarmno for Axis (62 Byte)
//Offset 182
   ZInfo0 : ARRAY  [0 .. 63 ] OF WORD ;	//Additional Value for UserAlarms 700000 to 700063
//Offset 310
   ChanA : ARRAY  [1 .. 10 ] OF STRUCT 	//From Channel 1 to Channel 10
    FDD_5C00xx : ARRAY  [0 .. 15 ] OF //Feed disable A.no.51000-510015
    BOOL ;
    FDD_RID_5C01xx : ARRAY  [0 .. 31 ] OF //Feed and read-in disable A.no.510100-510131
    BOOL ;
    RID_5C02xx : ARRAY  [0 .. 31 ] OF //Read-in disable A.no.510200-510231
    BOOL ;
    NCSD_5C03xx : ARRAY  [0 .. 15 ] OF //NC start disable A.no.510300-510315
    BOOL ;
    FdStop_1_5C11xx : ARRAY  [0 .. 15 ] OF //Feed stop GEOaxis 1 A.no.511100-511115
    BOOL ;
    FdStop_2_5C12xx : ARRAY  [0 .. 15 ] OF //Feed stop GEOaxis 2 A.no.511200-511215
    BOOL ;
    FdStop_3_5C13xx : ARRAY  [0 .. 15 ] OF //Feed stop GEOaxis 3 A.no.511300-511315
    BOOL ;
   END_STRUCT ;	//Alarmno for Chan are 5Cxxxx; C is the ChannelNo, except Channel 10. Channel 10
   AxisA : ARRAY  [1 .. 32 ] OF STRUCT 	//From Axis 1 to Axis 31
    AAFdStop60AAxx : ARRAY  [0 .. 15 ] OF //Feed stop axis/spindle
    BOOL ;
   END_STRUCT ;	//Alarmno for Axis are 60AAxx; A is the Axisno.
//Offset 554
   UserA : ARRAY  [0 .. 31 ] OF STRUCT
    A70UUxx : ARRAY  [0 .. 63 ] OF //Alarm 700000-700063 (user area 0)
    BOOL ;
   END_STRUCT ;	//Alarmno for UserAlarms are 7yUUxx; U is the Userarea, y = Db1004.UserDek2No[U]
  END_STRUCT ;	
END_TYPE

TYPE UDT 1071
VERSION : 0.0
  STRUCT
   MTIF : ARRAY  [1 .. 16 ] OF STRUCT
    MtType : INT ;
    MtPlaces : INT ;
    MtDistance : REAL ;
    MtNum : INT ;	// MT-No. to be positioned to
    MtPlaceNum : INT ;	// MT-PlaceNo. ~
    ToolHolder : INT ;	// TH-No as reference for MT-positioning
    IF : ARRAY  [1 .. 3 ] OF STRUCT
     reserved : INT ;	// reserved
    END_STRUCT ;
   END_STRUCT ;
  END_STRUCT ;	
END_TYPE

TYPE UDT 1072
VERSION : 0.0
  STRUCT
   MTIF : ARRAY  [1 .. 16 ] OF STRUCT
    MtType : INT ;
    MtPlaces : INT ;
    MtDistance : REAL ;
    MtNumNew : INT ;	// MT-No. new Tool
    MtPlaceNumNew : INT ;	// MtoolPlaceNum  ~
    MtNumOld : INT ;	// MT-No. old Tool
    MtPlaceNumOld : INT ;	// MtoolPlaceNum  ~
    LocType : INT ;	//Tool new: location type
    SLeft : INT ;	//Tool new: size left
    SRight : INT ;	//Tool new: size right
    STop : INT ;	//Tool new: size top
    SBottom : INT ;	//Tool new: size bottom
    ToolInBuff : BOOL ;	//ID for tools in buffer
    IgnoreDisab : BOOL ;	//Ignore disabled
    TBUnloaded : BOOL ;	//To be unloaded
    TBLoaded : BOOL ;	//To be loaded
    MasterTool : BOOL ;	//Master tool
    n26_5 : BOOL ;	//reserved
    n26_6 : BOOL ;	//reserved
    HandTool : BOOL ;	//Hand tool
    ActTool : BOOL ;	//Active tool
    ToolEnabl : BOOL ;	//Tool enabled
    ToolDisab : BOOL ;	//Tool disabled
    Measured : BOOL ;	//Tool measured
    Prewarn : BOOL ;	//Prewarning limit reached
    ToolChange : BOOL ;	//Tool being changed
    FixedLoc : BOOL ;	//Tool fixed location coded
    ToolUsed : BOOL ;	//Tool was in use
    T_no : INT ;	//Tool new: T no.
    ToolHolder : INT ;	// TH-No as tool compensation reference
    MtMyMag : INT ;	// MtoolNumber the tool is loaded onto
    MtMyPlace : INT ;	// MtoolPlaceNum ~
    IF : ARRAY  [1 .. 7 ] OF STRUCT
     reserved : INT ;	// reserved
    END_STRUCT ;
   END_STRUCT ;
  END_STRUCT ;	
END_TYPE

TYPE UDT 1073
VERSION : 0.0
  STRUCT
   MTIF : ARRAY  [1 .. 16 ] OF STRUCT
    MtType : INT ;
    MtPlaces : INT ;
    MtDistance : REAL ;
    MtNumNew : INT ;	// MT-No. new Tool
    MtPlaceNumNew : INT ;	// MtoolPlaceNum  ~
    MtNumOld : INT ;	// MT-No. old Tool
    MtPlaceNumOld : INT ;	// MtoolPlaceNum  ~
    LocType : INT ;	//Tool new: location type
    SLeft : INT ;	//Tool new: size left
    SRight : INT ;	//Tool new: size right
    STop : INT ;	//Tool new: size top
    SBottom : INT ;	//Tool new: size bottom
    ToolInBuff : BOOL ;	//ID for tools in buffer
    IgnoreDisab : BOOL ;	//Ignore disabled
    TBUnloaded : BOOL ;	//To be unloaded
    TBLoaded : BOOL ;	//To be loaded
    MasterTool : BOOL ;	//Master tool
    n26_5 : BOOL ;	//reserved
    n26_6 : BOOL ;	//reserved
    HandTool : BOOL ;	//Hand tool
    ActTool : BOOL ;	//Active tool
    ToolEnabl : BOOL ;	//Tool enabled
    ToolDisab : BOOL ;	//Tool disabled
    Measured : BOOL ;	//Tool measured
    Prewarn : BOOL ;	//Prewarning limit reached
    ToolChange : BOOL ;	//Tool being changed
    FixedLoc : BOOL ;	//Tool fixed location coded
    ToolUsed : BOOL ;	//Tool was in use
    T_no : INT ;	//Tool new: T no.
    ToolHolder : INT ;	// TH-No as tool compensation reference
    MtMyMag : INT ;	// MtoolNumber the tool is loaded onto
    MtMyPlace : INT ;	// MtoolPlaceNum ~
    IF : ARRAY  [1 .. 7 ] OF STRUCT
     reserved : INT ;	// reserved
    END_STRUCT ;
   END_STRUCT ;
  END_STRUCT ;	
END_TYPE

// FB 1: know-how protected block, not included

// FB 2: know-how protected block, not included

// FB 3: know-how protected block, not included

// FB 4: know-how protected block, not included

// FB 5: know-how protected block, not included

// FB 7: know-how protected block, not included

// FB 9: know-how protected block, not included

// FB 10: know-how protected block, not included

// FB 11: know-how protected block, not included

// FB 29: know-how protected block, not included

// FC 2: know-how protected block, not included

// FC 3: know-how protected block, not included

// FC 5: know-how protected block, not included

// FC 6: know-how protected block, not included

// FC 7: know-how protected block, not included

// FC 8: know-how protected block, not included

// FC 9: know-how protected block, not included

// FC 10: know-how protected block, not included

FUNCTION FC 12 : VOID
AUTHOR : NUMERIK
FAMILY : _800D
NAME : Basics
VERSION : 2.7
VAR_INPUT
  Chan : BYTE ;	//Index of Chan
END_VAR
BEGIN
// (block stored without names or comments; labels and parameter names are numbered)
END_FUNCTION

// FC 13: know-how protected block, not included

// FC 17: know-how protected block, not included

// FC 18: know-how protected block, not included

// FC 19: know-how protected block, not included

// FC 21: know-how protected block, not included

// FC 22: know-how protected block, not included

// FC 24: know-how protected block, not included

// FC 25: know-how protected block, not included

// FC 26: know-how protected block, not included

// FC 1005: know-how protected block, not included

// FC 1006: know-how protected block, not included

DATA_BLOCK DB 4
AUTHOR : NUMERIK
FAMILY : _800D
NAME : Basics
VERSION : 2.7
  STRUCT
   BOfeld0 : WORD  := W#16#CD54;	//Channel 1-8 ever 18 Bits
   BOfeld2 : WORD  := W#16#3553;
   BOfeld4 : WORD  := W#16#D54C;
   BOfeld6 : WORD  := W#16#5533;
   BOfeld8 : WORD  := W#16#55CD;
   BOfeld10 : WORD  := W#16#5435;
   BOfeld12 : WORD  := W#16#53D5;
   BOfeld14 : WORD  := W#16#4C55;
   BOfeld16 : WORD  := W#16#3355;
   BOfeld18 : WORD  := W#16#5555;	//18 Axes/Spindles ever 2 Bit
   BOfeld20 : WORD  := W#16#5555;
   BOfeld22 : WORD  := W#16#F5F0;	//10 User data area ever 8 Bit (Begin: DBB23)
   BOfeld24 : WORD  := W#16#F0F0;
   BOfeld26 : WORD  := W#16#F0F0;
   BOfeld28 : WORD  := W#16#F0F0;
   BOfeld30 : WORD  := W#16#F0F0;
   BOfeld32 : WORD  := W#16#F0F0;
   BOfeld34 : WORD  := W#16#F0F0;
   BOfeld36 : WORD  := W#16#F0F0;
   BOfeld38 : WORD  := W#16#F0F0;
   BOfeld40 : WORD  := W#16#F0F0;
   BOfeld42 : WORD  := W#16#F0F0;
   BOfeld44 : WORD  := W#16#F0F0;
   BOfeld46 : WORD  := W#16#F0F0;
   BOfeld48 : WORD  := W#16#F0F0;
   BOfeld50 : WORD  := W#16#F0F0;
   BOfeld52 : WORD  := W#16#F0F0;
   BOfeld54 : WORD  := W#16#F0F0;
   BOfeld56 : WORD  := W#16#F0F0;
   BOfeld58 : WORD  := W#16#F0F0;
   BOfeld60 : WORD  := W#16#F0F0;
   BOfeld62 : BYTE  := B#16#F0;
   NumUser : BYTE  := B#16#A;
   maganz : BYTE ;	//for TM, number of Magazine
   wzv : BYTE ;
   wzvdat : ARRAY  [1 .. 160 ] OF BYTE ;	//32 Magazine, possibly ever 5 Byte + Spindle
  END_STRUCT ;	
BEGIN
   BOfeld0 := W#16#CD54;
   BOfeld2 := W#16#3553;
   BOfeld4 := W#16#D54C;
   BOfeld6 := W#16#5533;
   BOfeld8 := W#16#55CD;
   BOfeld10 := W#16#5435;
   BOfeld12 := W#16#53D5;
   BOfeld14 := W#16#4C55;
   BOfeld16 := W#16#3355;
   BOfeld18 := W#16#5555;
   BOfeld20 := W#16#5555;
   BOfeld22 := W#16#F5F0;
   BOfeld24 := W#16#F0F0;
   BOfeld26 := W#16#F0F0;
   BOfeld28 := W#16#F0F0;
   BOfeld30 := W#16#F0F0;
   BOfeld32 := W#16#F0F0;
   BOfeld34 := W#16#F0F0;
   BOfeld36 := W#16#F0F0;
   BOfeld38 := W#16#F0F0;
   BOfeld40 := W#16#F0F0;
   BOfeld42 := W#16#F0F0;
   BOfeld44 := W#16#F0F0;
   BOfeld46 := W#16#F0F0;
   BOfeld48 := W#16#F0F0;
   BOfeld50 := W#16#F0F0;
   BOfeld52 := W#16#F0F0;
   BOfeld54 := W#16#F0F0;
   BOfeld56 := W#16#F0F0;
   BOfeld58 := W#16#F0F0;
   BOfeld60 := W#16#F0F0;
   BOfeld62 := B#16#F0;
   NumUser := B#16#A;
END_DATA_BLOCK

DATA_BLOCK DB 5
AUTHOR : NUMERIK
FAMILY : _800D
NAME : Basics
VERSION : 2.7
  STRUCT
   Ch1_DB2_310 : BOOL  := TRUE;	// (Channel 1-10 ever 18 Bits):  error message
   Ch1_DB2_311 : BOOL ;	// Channel 1, DB2.DBB311; operational message
   Ch1_DB2_312 : BOOL  := TRUE;	// Channel 1, DB2.DBB312; error message
   Ch1_DB2_313 : BOOL  := TRUE;	// error message
   Ch1_DB2_314 : BOOL ;	// operational message
   Ch1_DB2_315 : BOOL ;	// operational message
   Ch1_DB2_316 : BOOL  := TRUE;	// error message
   Ch1_DB2_317 : BOOL  := TRUE;	// error message
   Ch1_DB2_318 : BOOL ;	// operational message
   Ch1_DB2_319 : BOOL ;	// operational message
   Ch1_DB2_320 : BOOL  := TRUE;	// error message
   Ch1_DB2_321 : BOOL ;	// operational message
   Ch1_DB2_322 : BOOL  := TRUE;	// error message
   Ch1_DB2_323 : BOOL ;	// operational message
   Ch1_DB2_324 : BOOL  := TRUE;	// error message
   Ch1_DB2_325 : BOOL ;	// operational message
   Ch1_DB2_326 : BOOL  := TRUE;	// error message
   Ch1_DB2_327 : BOOL ;	// operational message
   Ch2_DB2_328 : BOOL  := TRUE;	// Channel 2, DB2.DBB328; error message
   Ch2_DB2_329 : BOOL ;	// Channel 2, DB2.DBB329; operational message
   Ch2_DB2_330 : BOOL  := TRUE;	// error message
   Ch2_DB2_331 : BOOL  := TRUE;	// error message
   Ch2_DB2_332 : BOOL ;	// operational message
   Ch2_DB2_333 : BOOL ;	// operational message
   Ch2_DB2_334 : BOOL  := TRUE;	// error message
   Ch2_DB2_335 : BOOL  := TRUE;	// error message
   Ch2_DB2_336 : BOOL ;	// operational message
   Ch2_DB2_337 : BOOL ;	// operational message
   Ch2_DB2_338 : BOOL  := TRUE;	// error message
   Ch2_DB2_339 : BOOL ;	// operational message
   Ch2_DB2_340 : BOOL  := TRUE;	// error message
   Ch2_DB2_341 : BOOL ;	// operational message
   Ch2_DB2_342 : BOOL  := TRUE;	// error message
   Ch2_DB2_343 : BOOL ;	// operational message
   Ch2_DB2_344 : BOOL  := TRUE;	// error message
   Ch2_DB2_345 : BOOL ;	// operational message
   Ch3_DB2_346 : BOOL  := TRUE;	// Channel 3, DB2.DBB346; error message
   Ch3_DB2_347 : BOOL ;	// Channel 3, DB2.DBB347; operational message
   Ch3_DB2_348 : BOOL  := TRUE;	// error message
   Ch3_DB2_349 : BOOL  := TRUE;	// error message
   Ch3_DB2_350 : BOOL ;	// operational message
   Ch3_DB2_351 : BOOL ;	// operational message
   Ch3_DB2_352 : BOOL  := TRUE;	// error message
   Ch3_DB2_353 : BOOL  := TRUE;	// error message
   Ch3_DB2_354 : BOOL ;	// operational message
   Ch3_DB2_355 : BOOL ;	// operational message
   Ch3_DB2_356 : BOOL  := TRUE;	// error message
   Ch3_DB2_357 : BOOL ;	// operational message
   Ch3_DB2_358 : BOOL  := TRUE;	// error message
   Ch3_DB2_359 : BOOL ;	// operational message
   Ch3_DB2_360 : BOOL  := TRUE;	// error message
   Ch3_DB2_361 : BOOL ;	// operational message
   Ch3_DB2_362 : BOOL  := TRUE;	// error message
   Ch3_DB2_363 : BOOL ;	// operational message
   Ch4_DB2_364 : BOOL  := TRUE;	// Channel 4, DB2.DBB364; error message
   Ch4_DB2_365 : BOOL ;	// Channel 4, DB2.DBB365; operational message
   Ch4_DB2_366 : BOOL  := TRUE;	// error message
   Ch4_DB2_367 : BOOL  := TRUE;	// error message
   Ch4_DB2_368 : BOOL ;	// operational message
   Ch4_DB2_369 : BOOL ;	// operational message
   Ch4_DB2_370 : BOOL  := TRUE;	// error message
   Ch4_DB2_371 : BOOL  := TRUE;	// error message
   Ch4_DB2_372 : BOOL ;	// operational message
   Ch4_DB2_373 : BOOL ;	// operational message
   Ch4_DB2_374 : BOOL  := TRUE;	// error message
   Ch4_DB2_375 : BOOL ;	// operational message
   Ch4_DB2_376 : BOOL  := TRUE;	// error message
   Ch4_DB2_377 : BOOL ;	// operational message
   Ch4_DB2_378 : BOOL  := TRUE;	// error message
   Ch4_DB2_379 : BOOL ;	// operational message
   Ch4_DB2_380 : BOOL  := TRUE;	// error message
   Ch4_DB2_381 : BOOL ;	// operational message
   Ch5_DB2_382 : BOOL  := TRUE;	// Channel 5, DB2.DBB382; error message
   Ch5_DB2_383 : BOOL ;	// Channel 5, DB2.DBB383; operational message
   Ch5_DB2_384 : BOOL  := TRUE;	// error message
   Ch5_DB2_385 : BOOL  := TRUE;	// error message
   Ch5_DB2_386 : BOOL ;	// operational message
   Ch5_DB2_387 : BOOL ;	// operational message
   Ch5_DB2_388 : BOOL  := TRUE;	// error message
   Ch5_DB2_389 : BOOL  := TRUE;	// error message
   Ch5_DB2_390 : BOOL ;	// operational message
   Ch5_DB2_391 : BOOL ;	// operational message
   Ch5_DB2_392 : BOOL  := TRUE;	// error message
   Ch5_DB2_393 : BOOL ;	// operational message
   Ch5_DB2_394 : BOOL  := TRUE;	// error message
   Ch5_DB2_395 : BOOL ;	// operational message
   Ch5_DB2_396 : BOOL  := TRUE;	// error message
   Ch5_DB2_397 : BOOL ;	// operational message
   Ch5_DB2_398 : BOOL  := TRUE;	// error message
   Ch5_DB2_399 : BOOL ;	// operational message
   Ch6_DB2_400 : BOOL  := TRUE;	// Channel 6, DB2.DBB400; error message
   Ch6_DB2_401 : BOOL ;	// Channel 6, DB2.DBB401; operational message
   Ch6_DB2_402 : BOOL  := TRUE;	// error message
   Ch6_DB2_403 : BOOL  := TRUE;	// error message
   Ch6_DB2_404 : BOOL ;	// operational message
   Ch6_DB2_405 : BOOL ;	// operational message
   Ch6_DB2_406 : BOOL  := TRUE;	// error message
   Ch6_DB2_407 : BOOL  := TRUE;	// error message
   Ch6_DB2_408 : BOOL ;	// operational message
   Ch6_DB2_409 : BOOL ;	// operational message
   Ch6_DB2_410 : BOOL  := TRUE;	// error message
   Ch6_DB2_411 : BOOL ;	// operational message
   Ch6_DB2_412 : BOOL  := TRUE;	// error message
   Ch6_DB2_413 : BOOL ;	// operational message
   Ch6_DB2_414 : BOOL  := TRUE;	// error message
   Ch6_DB2_415 : BOOL ;	// operational message
   Ch6_DB2_416 : BOOL  := TRUE;	// error message
   Ch6_DB2_417 : BOOL ;	// operational message
   Ch7_DB2_418 : BOOL  := TRUE;	// Channel 7, DB2.DBB418; error message
   Ch7_DB2_419 : BOOL ;	// Channel 7, DB2.DBB419; operational message
   Ch7_DB2_420 : BOOL  := TRUE;	// error message
   Ch7_DB2_421 : BOOL  := TRUE;	// error message
   Ch7_DB2_422 : BOOL ;	// operational message
   Ch7_DB2_423 : BOOL ;	// operational message
   Ch7_DB2_424 : BOOL  := TRUE;	// error message
   Ch7_DB2_425 : BOOL  := TRUE;	// error message
   Ch7_DB2_426 : BOOL ;	// operational message
   Ch7_DB2_427 : BOOL ;	// operational message
   Ch7_DB2_428 : BOOL  := TRUE;	// error message
   Ch7_DB2_429 : BOOL ;	// operational message
   Ch7_DB2_430 : BOOL  := TRUE;	// error message
   Ch7_DB2_431 : BOOL ;	// operational message
   Ch7_DB2_432 : BOOL  := TRUE;	// error message
   Ch7_DB2_433 : BOOL ;	// operational message
   Ch7_DB2_434 : BOOL  := TRUE;	// error message
   Ch7_DB2_435 : BOOL ;	// operational message
   Ch8_DB2_436 : BOOL  := TRUE;	// Channel 8, DB2.DBB436; error message
   Ch8_DB2_437 : BOOL ;	// Channel 8, DB2.DBB437; operational message
   Ch8_DB2_438 : BOOL  := TRUE;	// error message
   Ch8_DB2_439 : BOOL  := TRUE;	// error message
   Ch8_DB2_440 : BOOL ;	// operational message
   Ch8_DB2_441 : BOOL ;	// operational message
   Ch8_DB2_442 : BOOL  := TRUE;	// error message
   Ch8_DB2_443 : BOOL  := TRUE;	// error message
   Ch8_DB2_444 : BOOL ;	// operational message
   Ch8_DB2_445 : BOOL ;	// operational message
   Ch8_DB2_446 : BOOL  := TRUE;	// error message
   Ch8_DB2_447 : BOOL ;	// operational message
   Ch8_DB2_448 : BOOL  := TRUE;	// error message
   Ch8_DB2_449 : BOOL ;	// operational message
   Ch8_DB2_450 : BOOL  := TRUE;	// error message
   Ch8_DB2_451 : BOOL ;	// operational message
   Ch8_DB2_452 : BOOL  := TRUE;	// error message
   Ch8_DB2_453 : BOOL ;	// operational message
   Ch9_DB2_454 : BOOL  := TRUE;	// Channel 9, DB2.DBB454; error message
   Ch9_DB2_455 : BOOL ;	// Channel 9, DB2.DBB455; operational message
   Ch9_DB2_456 : BOOL  := TRUE;	// error message
   Ch9_DB2_457 : BOOL  := TRUE;	// error message
   Ch9_DB2_458 : BOOL ;	// operational message
   Ch9_DB2_459 : BOOL ;	// operational message
   Ch9_DB2_460 : BOOL  := TRUE;	// error message
   Ch9_DB2_461 : BOOL  := TRUE;	// error message
   Ch9_DB2_462 : BOOL ;	// operational message
   Ch9_DB2_463 : BOOL ;	// operational message
   Ch9_DB2_464 : BOOL  := TRUE;	// error message
   Ch9_DB2_465 : BOOL ;	// operational message
   Ch9_DB2_466 : BOOL  := TRUE;	// error message
   Ch9_DB2_467 : BOOL ;	// operational message
   Ch9_DB2_468 : BOOL  := TRUE;	// error message
   Ch9_DB2_469 : BOOL ;	// operational message
   Ch9_DB2_470 : BOOL  := TRUE;	// error message
   Ch9_DB2_471 : BOOL ;	// operational message
   Ch10_DB2_472 : BOOL  := TRUE;	// Channel 10, DB2.DBB472; error message
   Ch10_DB2_473 : BOOL ;	// Channel 10, DB2.DBB473; operational message
   Ch10_DB2_474 : BOOL  := TRUE;	// error message
   Ch10_DB2_475 : BOOL  := TRUE;	// error message
   Ch10_DB2_476 : BOOL ;	// operational message
   Ch10_DB2_477 : BOOL ;	// operational message
   Ch10_DB2_478 : BOOL  := TRUE;	// error message
   Ch10_DB2_479 : BOOL  := TRUE;	// error message
   Ch10_DB2_480 : BOOL ;	// operational message
   Ch10_DB2_481 : BOOL ;	// operational message
   Ch10_DB2_482 : BOOL  := TRUE;	// error message
   Ch10_DB2_483 : BOOL ;	// operational message
   Ch10_DB2_484 : BOOL  := TRUE;	// error message
   Ch10_DB2_485 : BOOL ;	// operational message
   Ch10_DB2_486 : BOOL  := TRUE;	// error message
   Ch10_DB2_487 : BOOL ;	// operational message
   Ch10_DB2_488 : BOOL  := TRUE;	// error message
   Ch10_DB2_489 : BOOL ;	// operational message
   Ax1_DB2_490 : BOOL  := TRUE;	// (32 Axes/Spindles ever 2 Bit):  error message
   Ax1_DB2_491 : BOOL ;	// Axis 1, DB2.DBB491; operational message
   Ax2_DB2_492 : BOOL  := TRUE;	// Axis 2, DB2.DBB492; error message
   Ax2_DB2_493 : BOOL ;	// Axis 2, DB2.DBB493; operational message
   Ax3_DB2_494 : BOOL  := TRUE;	// error message
   Ax3_DB2_495 : BOOL ;	// operational message
   Ax4_DB2_496 : BOOL  := TRUE;	// error message
   Ax4_DB2_497 : BOOL ;	// operational message
   Ax5_DB2_498 : BOOL  := TRUE;	// error message
   Ax5_DB2_499 : BOOL ;	// operational message
   Ax6_DB2_500 : BOOL  := TRUE;	// error message
   Ax6_DB2_501 : BOOL ;	// operational message
   Ax7_DB2_502 : BOOL  := TRUE;	// error message
   Ax7_DB2_503 : BOOL ;	// operational message
   Ax8_DB2_504 : BOOL  := TRUE;	// error message
   Ax8_DB2_505 : BOOL ;	// operational message
   Ax9_DB2_506 : BOOL  := TRUE;	// error message
   Ax9_DB2_507 : BOOL ;	// operational message
   Ax10_DB2_508 : BOOL  := TRUE;	// error message
   Ax10_DB2_509 : BOOL ;	// operational message
   Ax11_DB2_510 : BOOL  := TRUE;	// error message
   Ax11_DB2_511 : BOOL ;	// operational message
   Ax12_DB2_512 : BOOL  := TRUE;	// error message
   Ax12_DB2_513 : BOOL ;	// operational message
   Ax13_DB2_514 : BOOL  := TRUE;	// error message
   Ax13_DB2_515 : BOOL ;	// operational message
   Ax14_DB2_516 : BOOL  := TRUE;	// error message
   Ax14_DB2_517 : BOOL ;	// operational message
   Ax15_DB2_518 : BOOL  := TRUE;	// error message
   Ax15_DB2_519 : BOOL ;	// operational message
   Ax16_DB2_520 : BOOL  := TRUE;	// error message
   Ax16_DB2_521 : BOOL ;	// operational message
   Ax17_DB2_522 : BOOL  := TRUE;	// error message
   Ax17_DB2_523 : BOOL ;	// operational message
   Ax18_DB2_524 : BOOL  := TRUE;	// error message
   Ax18_DB2_525 : BOOL ;	// operational message
   Ax19_DB2_526 : BOOL  := TRUE;	// error message
   Ax19_DB2_527 : BOOL ;	// operational message
   Ax20_DB2_528 : BOOL  := TRUE;	// error message
   Ax20_DB2_529 : BOOL ;	// operational message
   Ax21_DB2_530 : BOOL  := TRUE;	// error message
   Ax21_DB2_531 : BOOL ;	// operational message
   Ax22_DB2_532 : BOOL  := TRUE;	// error message
   Ax22_DB2_533 : BOOL ;	// operational message
   Ax23_DB2_534 : BOOL  := TRUE;	// error message
   Ax23_DB2_535 : BOOL ;	// operational message
   Ax24_DB2_536 : BOOL  := TRUE;	// error message
   Ax24_DB2_537 : BOOL ;	// operational message
   Ax25_DB2_538 : BOOL  := TRUE;	// error message
   Ax25_DB2_539 : BOOL ;	// operational message
   Ax26_DB2_540 : BOOL  := TRUE;	// error message
   Ax26_DB2_541 : BOOL ;	// operational message
   Ax27_DB2_542 : BOOL  := TRUE;	// error message
   Ax27_DB2_543 : BOOL ;	// operational message
   Ax28_DB2_544 : BOOL  := TRUE;	// error message
   Ax28_DB2_545 : BOOL ;	// operational message
   Ax29_DB2_546 : BOOL  := TRUE;	// error message
   Ax29_DB2_547 : BOOL ;	// operational message
   Ax30_DB2_548 : BOOL  := TRUE;	// error message
   Ax30_DB2_549 : BOOL ;	// operational message
   Ax31_DB2_550 : BOOL  := TRUE;	// error message
   Ax31_DB2_551 : BOOL ;	// operational message
   Ax32_DB2_552 : BOOL  := TRUE;	// error message
   Ax32_DB2_553 : BOOL ;	// operational message
   User0_DB2_554 : BOOL  := TRUE;	// (32 User data area ever 8 Bit):  error message
   User0_DB2_555 : BOOL  := TRUE;	// UserDataArea 0, DB2.DBB555; error message
   User0_DB2_556 : BOOL  := TRUE;	// error message
   User0_DB2_557 : BOOL  := TRUE;	// error message
   User0_DB2_558 : BOOL ;	// operational message
   User0_DB2_559 : BOOL ;	// operational message
   User0_DB2_560 : BOOL ;	// operational message
   User0_DB2_561 : BOOL ;	// operational message
   User1_DB2_562 : BOOL  := TRUE;	// UserDataArea 1, DB2.DBB562; error message
   User1_DB2_563 : BOOL  := TRUE;	// error message
   User1_DB2_564 : BOOL  := TRUE;	// error message
   User1_DB2_565 : BOOL  := TRUE;	// error message
   User1_DB2_566 : BOOL ;	// operational message
   User1_DB2_567 : BOOL ;	// operational message
   User1_DB2_568 : BOOL ;	// operational message
   User1_DB2_569 : BOOL ;	// operational message
   User2_DB2_570 : BOOL  := TRUE;	// UserDataArea 2, DB2.DBB570; error message
   User2_DB2_571 : BOOL  := TRUE;	// error message
   User2_DB2_572 : BOOL  := TRUE;	// error message
   User2_DB2_573 : BOOL  := TRUE;	// error message
   User2_DB2_574 : BOOL ;	// operational message
   User2_DB2_575 : BOOL ;	// operational message
   User2_DB2_576 : BOOL ;	// operational message
   User2_DB2_577 : BOOL ;	// operational message
   User3_DB2_578 : BOOL  := TRUE;	// UserDataArea 3, DB2.DBB578; error message
   User3_DB2_579 : BOOL  := TRUE;	// error message
   User3_DB2_580 : BOOL  := TRUE;	// error message
   User3_DB2_581 : BOOL  := TRUE;	// error message
   User3_DB2_582 : BOOL ;	// operational message
   User3_DB2_583 : BOOL ;	// operational message
   User3_DB2_584 : BOOL ;	// operational message
   User3_DB2_585 : BOOL ;	// operational message
   User4_DB2_586 : BOOL  := TRUE;	// UserDataArea 4, DB2.DBB586; error message
   User4_DB2_587 : BOOL  := TRUE;	// error message
   User4_DB2_588 : BOOL  := TRUE;	// error message
   User4_DB2_589 : BOOL  := TRUE;	// error message
   User4_DB2_590 : BOOL ;	// operational message
   User4_DB2_591 : BOOL ;	// operational message
   User4_DB2_592 : BOOL ;	// operational message
   User4_DB2_593 : BOOL ;	// operational message
   User5_DB2_594 : BOOL  := TRUE;	// UserDataArea 5, DB2.DBB594; error message
   User5_DB2_595 : BOOL  := TRUE;	// error message
   User5_DB2_596 : BOOL  := TRUE;	// error message
   User5_DB2_597 : BOOL  := TRUE;	// error message
   User5_DB2_598 : BOOL ;	// operational message
   User5_DB2_599 : BOOL ;	// operational message
   User5_DB2_600 : BOOL ;	// operational message
   User5_DB2_601 : BOOL ;	// operational message
   User6_DB2_602 : BOOL  := TRUE;	// UserDataArea 6, DB2.DBB602; error message
   User6_DB2_603 : BOOL  := TRUE;	// error message
   User6_DB2_604 : BOOL  := TRUE;	// error message
   User6_DB2_605 : BOOL  := TRUE;	// error message
   User6_DB2_606 : BOOL ;	// operational message
   User6_DB2_607 : BOOL ;	// operational message
   User6_DB2_608 : BOOL ;	// operational message
   User6_DB2_609 : BOOL ;	// operational message
   User7_DB2_610 : BOOL  := TRUE;	// UserDataArea 7, DB2.DBB610; error message
   User7_DB2_611 : BOOL  := TRUE;	// error message
   User7_DB2_612 : BOOL  := TRUE;	// error message
   User7_DB2_613 : BOOL  := TRUE;	// error message
   User7_DB2_614 : BOOL ;	// operational message
   User7_DB2_615 : BOOL ;	// operational message
   User7_DB2_616 : BOOL ;	// operational message
   User7_DB2_617 : BOOL ;	// operational message
   User8_DB2_618 : BOOL  := TRUE;	// UserDataArea 8, DB2.DBB618; error message
   User8_DB2_619 : BOOL  := TRUE;	// error message
   User8_DB2_620 : BOOL  := TRUE;	// error message
   User8_DB2_621 : BOOL  := TRUE;	// error message
   User8_DB2_622 : BOOL ;	// operational message
   User8_DB2_623 : BOOL ;	// operational message
   User8_DB2_624 : BOOL ;	// operational message
   User8_DB2_625 : BOOL ;	// operational message
   User9_DB2_626 : BOOL  := TRUE;	// UserDataArea 9, DB2.DBB626; error message
   User9_DB2_627 : BOOL  := TRUE;	// error message
   User9_DB2_628 : BOOL  := TRUE;	// error message
   User9_DB2_629 : BOOL  := TRUE;	// error message
   User9_DB2_630 : BOOL ;	// operational message
   User9_DB2_631 : BOOL ;	// operational message
   User9_DB2_632 : BOOL ;	// operational message
   User9_DB2_633 : BOOL ;	// operational message
   User10_DB2_634 : BOOL  := TRUE;	// UserDataArea 10, DB2.DBB634; error message
   User10_DB2_635 : BOOL  := TRUE;	// error message
   User10_DB2_636 : BOOL  := TRUE;	// error message
   User10_DB2_637 : BOOL  := TRUE;	// error message
   User10_DB2_638 : BOOL ;	// operational message
   User10_DB2_639 : BOOL ;	// operational message
   User10_DB2_640 : BOOL ;	// operational message
   User10_DB2_641 : BOOL ;	// operational message
   User11_DB2_642 : BOOL  := TRUE;	// UserDataArea 11, DB2.DBB642; error message
   User11_DB2_643 : BOOL  := TRUE;	// error message
   User11_DB2_644 : BOOL  := TRUE;	// error message
   User11_DB2_645 : BOOL  := TRUE;	// error message
   User11_DB2_646 : BOOL ;	// operational message
   User11_DB2_647 : BOOL ;	// operational message
   User11_DB2_648 : BOOL ;	// operational message
   User11_DB2_649 : BOOL ;	// operational message
   User12_DB2_650 : BOOL  := TRUE;	// UserDataArea 12, DB2.DBB650; error message
   User12_DB2_651 : BOOL  := TRUE;	// error message
   User12_DB2_652 : BOOL  := TRUE;	// error message
   User12_DB2_653 : BOOL  := TRUE;	// error message
   User12_DB2_654 : BOOL ;	// operational message
   User12_DB2_655 : BOOL ;	// operational message
   User12_DB2_656 : BOOL ;	// operational message
   User12_DB2_657 : BOOL ;	// operational message
   User13_DB2_658 : BOOL  := TRUE;	// UserDataArea 13, DB2.DBB658; error message
   User13_DB2_659 : BOOL  := TRUE;	// error message
   User13_DB2_660 : BOOL  := TRUE;	// error message
   User13_DB2_661 : BOOL  := TRUE;	// error message
   User13_DB2_662 : BOOL ;	// operational message
   User13_DB2_663 : BOOL ;	// operational message
   User13_DB2_664 : BOOL ;	// operational message
   User13_DB2_665 : BOOL ;	// operational message
   User14_DB2_666 : BOOL  := TRUE;	// UserDataArea 14, DB2.DBB666; error message
   User14_DB2_667 : BOOL  := TRUE;	// error message
   User14_DB2_668 : BOOL  := TRUE;	// error message
   User14_DB2_669 : BOOL  := TRUE;	// error message
   User14_DB2_670 : BOOL ;	// operational message
   User14_DB2_671 : BOOL ;	// operational message
   User14_DB2_672 : BOOL ;	// operational message
   User14_DB2_673 : BOOL ;	// operational message
   User15_DB2_674 : BOOL  := TRUE;	// UserDataArea 15, DB2.DBB674; error message
   User15_DB2_675 : BOOL  := TRUE;	// error message
   User15_DB2_676 : BOOL  := TRUE;	// error message
   User15_DB2_677 : BOOL  := TRUE;	// error message
   User15_DB2_678 : BOOL ;	// operational message
   User15_DB2_679 : BOOL ;	// operational message
   User15_DB2_680 : BOOL ;	// operational message
   User15_DB2_681 : BOOL ;	// operational message
   User16_DB2_682 : BOOL  := TRUE;	// UserDataArea 16, DB2.DBB682; error message
   User16_DB2_683 : BOOL  := TRUE;	// error message
   User16_DB2_684 : BOOL  := TRUE;	// error message
   User16_DB2_685 : BOOL  := TRUE;	// error message
   User16_DB2_686 : BOOL ;	// operational message
   User16_DB2_687 : BOOL ;	// operational message
   User16_DB2_688 : BOOL ;	// operational message
   User16_DB2_689 : BOOL ;	// operational message
   User17_DB2_690 : BOOL  := TRUE;	// UserDataArea 17, DB2.DBB690; error message
   User17_DB2_691 : BOOL  := TRUE;	// error message
   User17_DB2_692 : BOOL  := TRUE;	// error message
   User17_DB2_693 : BOOL  := TRUE;	// error message
   User17_DB2_694 : BOOL ;	// operational message
   User17_DB2_695 : BOOL ;	// operational message
   User17_DB2_696 : BOOL ;	// operational message
   User17_DB2_697 : BOOL ;	// operational message
   User18_DB2_698 : BOOL  := TRUE;	// UserDataArea 18, DB2.DBB698; error message
   User18_DB2_699 : BOOL  := TRUE;	// error message
   User18_DB2_700 : BOOL  := TRUE;	// error message
   User18_DB2_701 : BOOL  := TRUE;	// error message
   User18_DB2_702 : BOOL ;	// operational message
   User18_DB2_703 : BOOL ;	// operational message
   User18_DB2_704 : BOOL ;	// operational message
   User18_DB2_705 : BOOL ;	// operational message
   User19_DB2_706 : BOOL  := TRUE;	// UserDataArea 19, DB2.DBB706; error message
   User19_DB2_707 : BOOL  := TRUE;	// error message
   User19_DB2_708 : BOOL  := TRUE;	// error message
   User19_DB2_709 : BOOL  := TRUE;	// error message
   User19_DB2_710 : BOOL ;	// operational message
   User19_DB2_711 : BOOL ;	// operational message
   User19_DB2_712 : BOOL ;	// operational message
   User19_DB2_713 : BOOL ;	// operational message
   User20_DB2_714 : BOOL  := TRUE;	// UserDataArea 20, DB2.DBB714; error message
   User20_DB2_715 : BOOL  := TRUE;	// error message
   User20_DB2_716 : BOOL  := TRUE;	// error message
   User20_DB2_717 : BOOL  := TRUE;	// error message
   User20_DB2_718 : BOOL ;	// operational message
   User20_DB2_719 : BOOL ;	// operational message
   User20_DB2_720 : BOOL ;	// operational message
   User20_DB2_721 : BOOL ;	// operational message
   User21_DB2_722 : BOOL  := TRUE;	// UserDataArea 21, DB2.DBB722; error message
   User21_DB2_723 : BOOL  := TRUE;	// error message
   User21_DB2_724 : BOOL  := TRUE;	// error message
   User21_DB2_725 : BOOL  := TRUE;	// error message
   User21_DB2_726 : BOOL ;	// operational message
   User21_DB2_727 : BOOL ;	// operational message
   User21_DB2_728 : BOOL ;	// operational message
   User21_DB2_729 : BOOL ;	// operational message
   User22_DB2_730 : BOOL  := TRUE;	// UserDataArea 22, DB2.DBB730; error message
   User22_DB2_731 : BOOL  := TRUE;	// error message
   User22_DB2_732 : BOOL  := TRUE;	// error message
   User22_DB2_733 : BOOL  := TRUE;	// error message
   User22_DB2_734 : BOOL ;	// operational message
   User22_DB2_735 : BOOL ;	// operational message
   User22_DB2_736 : BOOL ;	// operational message
   User22_DB2_737 : BOOL ;	// operational message
   User23_DB2_738 : BOOL  := TRUE;	// UserDataArea 23, DB2.DBB738; error message
   User23_DB2_739 : BOOL  := TRUE;	// error message
   User23_DB2_740 : BOOL  := TRUE;	// error message
   User23_DB2_741 : BOOL  := TRUE;	// error message
   User23_DB2_742 : BOOL ;	// operational message
   User23_DB2_743 : BOOL ;	// operational message
   User23_DB2_744 : BOOL ;	// operational message
   User23_DB2_745 : BOOL ;	// operational message
   User24_DB2_746 : BOOL  := TRUE;	// UserDataArea 24, DB2.DBB746; error message
   User24_DB2_747 : BOOL  := TRUE;	// error message
   User24_DB2_748 : BOOL  := TRUE;	// error message
   User24_DB2_749 : BOOL  := TRUE;	// error message
   User24_DB2_750 : BOOL ;	// operational message
   User24_DB2_751 : BOOL ;	// operational message
   User24_DB2_752 : BOOL ;	// operational message
   User24_DB2_753 : BOOL ;	// operational message
   User25_DB2_754 : BOOL  := TRUE;	// UserDataArea 25, DB2.DBB754; error message
   User25_DB2_755 : BOOL  := TRUE;	// error message
   User25_DB2_756 : BOOL  := TRUE;	// error message
   User25_DB2_757 : BOOL  := TRUE;	// error message
   User25_DB2_758 : BOOL ;	// operational message
   User25_DB2_759 : BOOL ;	// operational message
   User25_DB2_760 : BOOL ;	// operational message
   User25_DB2_761 : BOOL ;	// operational message
   User26_DB2_762 : BOOL  := TRUE;	// UserDataArea 26, DB2.DBB762; error message
   User26_DB2_763 : BOOL  := TRUE;	// error message
   User26_DB2_764 : BOOL  := TRUE;	// error message
   User26_DB2_765 : BOOL  := TRUE;	// error message
   User26_DB2_766 : BOOL ;	// operational message
   User26_DB2_767 : BOOL ;	// operational message
   User26_DB2_768 : BOOL ;	// operational message
   User26_DB2_769 : BOOL ;	// operational message
   User27_DB2_770 : BOOL  := TRUE;	// UserDataArea 27, DB2.DBB770; error message
   User27_DB2_771 : BOOL  := TRUE;	// error message
   User27_DB2_772 : BOOL  := TRUE;	// error message
   User27_DB2_773 : BOOL  := TRUE;	// error message
   User27_DB2_774 : BOOL ;	// operational message
   User27_DB2_775 : BOOL ;	// operational message
   User27_DB2_776 : BOOL ;	// operational message
   User27_DB2_777 : BOOL ;	// operational message
   User28_DB2_778 : BOOL  := TRUE;	// UserDataArea 28, DB2.DBB778; error message
   User28_DB2_779 : BOOL  := TRUE;	// error message
   User28_DB2_780 : BOOL  := TRUE;	// error message
   User28_DB2_781 : BOOL  := TRUE;	// error message
   User28_DB2_782 : BOOL ;	// operational message
   User28_DB2_783 : BOOL ;	// operational message
   User28_DB2_784 : BOOL ;	// operational message
   User28_DB2_785 : BOOL ;	// operational message
   User29_DB2_786 : BOOL  := TRUE;	// UserDataArea 29, DB2.DBB786; error message
   User29_DB2_787 : BOOL  := TRUE;	// error message
   User29_DB2_788 : BOOL  := TRUE;	// error message
   User29_DB2_789 : BOOL  := TRUE;	// error message
   User29_DB2_790 : BOOL ;	// operational message
   User29_DB2_791 : BOOL ;	// operational message
   User29_DB2_792 : BOOL ;	// operational message
   User29_DB2_793 : BOOL ;	// operational message
   User30_DB2_794 : BOOL  := TRUE;	// UserDataArea 30, DB2.DBB794; error message
   User30_DB2_795 : BOOL  := TRUE;	// error message
   User30_DB2_796 : BOOL  := TRUE;	// error message
   User30_DB2_797 : BOOL  := TRUE;	// error message
   User30_DB2_798 : BOOL ;	// operational message
   User30_DB2_799 : BOOL ;	// operational message
   User30_DB2_800 : BOOL ;	// operational message
   User30_DB2_801 : BOOL ;	// operational message
   User31_DB2_802 : BOOL  := TRUE;	// UserDataArea 31, DB2.DBB802; error message
   User31_DB2_803 : BOOL  := TRUE;	// error message
   User31_DB2_804 : BOOL  := TRUE;	// error message
   User31_DB2_805 : BOOL  := TRUE;	// error message
   User31_DB2_806 : BOOL ;	// operational message
   User31_DB2_807 : BOOL ;	// operational message
   User31_DB2_808 : BOOL ;	// operational message
   User31_DB2_809 : BOOL ;	// operational message
   Bit62_4 : BOOL ;	// reserved
   Bit62_5 : BOOL ;	// reserved
   Bit62_6 : BOOL ;	// reserved
   Bit62_7 : BOOL ;	// reserved
   Byte63 : BYTE ;	// reserved
   Word64 : WORD ;	// reserved
   Word66 : WORD ;	// reserved
   Word68 : WORD ;	// reserved
   Word70 : WORD ;	// reserved
   UserDek2No : ARRAY  [0 .. 31 ] OF // UserDek2No: Value 0..9 possible
   BYTE  := B#16#0;
  END_STRUCT ;	
BEGIN
   Ch1_DB2_310 := TRUE;
   Ch1_DB2_312 := TRUE;
   Ch1_DB2_313 := TRUE;
   Ch1_DB2_316 := TRUE;
   Ch1_DB2_317 := TRUE;
   Ch1_DB2_320 := TRUE;
   Ch1_DB2_322 := TRUE;
   Ch1_DB2_324 := TRUE;
   Ch1_DB2_326 := TRUE;
   Ch2_DB2_328 := TRUE;
   Ch2_DB2_330 := TRUE;
   Ch2_DB2_331 := TRUE;
   Ch2_DB2_334 := TRUE;
   Ch2_DB2_335 := TRUE;
   Ch2_DB2_338 := TRUE;
   Ch2_DB2_340 := TRUE;
   Ch2_DB2_342 := TRUE;
   Ch2_DB2_344 := TRUE;
   Ch3_DB2_346 := TRUE;
   Ch3_DB2_348 := TRUE;
   Ch3_DB2_349 := TRUE;
   Ch3_DB2_352 := TRUE;
   Ch3_DB2_353 := TRUE;
   Ch3_DB2_356 := TRUE;
   Ch3_DB2_358 := TRUE;
   Ch3_DB2_360 := TRUE;
   Ch3_DB2_362 := TRUE;
   Ch4_DB2_364 := TRUE;
   Ch4_DB2_366 := TRUE;
   Ch4_DB2_367 := TRUE;
   Ch4_DB2_370 := TRUE;
   Ch4_DB2_371 := TRUE;
   Ch4_DB2_374 := TRUE;
   Ch4_DB2_376 := TRUE;
   Ch4_DB2_378 := TRUE;
   Ch4_DB2_380 := TRUE;
   Ch5_DB2_382 := TRUE;
   Ch5_DB2_384 := TRUE;
   Ch5_DB2_385 := TRUE;
   Ch5_DB2_388 := TRUE;
   Ch5_DB2_389 := TRUE;
   Ch5_DB2_392 := TRUE;
   Ch5_DB2_394 := TRUE;
   Ch5_DB2_396 := TRUE;
   Ch5_DB2_398 := TRUE;
   Ch6_DB2_400 := TRUE;
   Ch6_DB2_402 := TRUE;
   Ch6_DB2_403 := TRUE;
   Ch6_DB2_406 := TRUE;
   Ch6_DB2_407 := TRUE;
   Ch6_DB2_410 := TRUE;
   Ch6_DB2_412 := TRUE;
   Ch6_DB2_414 := TRUE;
   Ch6_DB2_416 := TRUE;
   Ch7_DB2_418 := TRUE;
   Ch7_DB2_420 := TRUE;
   Ch7_DB2_421 := TRUE;
   Ch7_DB2_424 := TRUE;
   Ch7_DB2_425 := TRUE;
   Ch7_DB2_428 := TRUE;
   Ch7_DB2_430 := TRUE;
   Ch7_DB2_432 := TRUE;
   Ch7_DB2_434 := TRUE;
   Ch8_DB2_436 := TRUE;
   Ch8_DB2_438 := TRUE;
   Ch8_DB2_439 := TRUE;
   Ch8_DB2_442 := TRUE;
   Ch8_DB2_443 := TRUE;
   Ch8_DB2_446 := TRUE;
   Ch8_DB2_448 := TRUE;
   Ch8_DB2_450 := TRUE;
   Ch8_DB2_452 := TRUE;
   Ch9_DB2_454 := TRUE;
   Ch9_DB2_456 := TRUE;
   Ch9_DB2_457 := TRUE;
   Ch9_DB2_460 := TRUE;
   Ch9_DB2_461 := TRUE;
   Ch9_DB2_464 := TRUE;
   Ch9_DB2_466 := TRUE;
   Ch9_DB2_468 := TRUE;
   Ch9_DB2_470 := TRUE;
   Ch10_DB2_472 := TRUE;
   Ch10_DB2_474 := TRUE;
   Ch10_DB2_475 := TRUE;
   Ch10_DB2_478 := TRUE;
   Ch10_DB2_479 := TRUE;
   Ch10_DB2_482 := TRUE;
   Ch10_DB2_484 := TRUE;
   Ch10_DB2_486 := TRUE;
   Ch10_DB2_488 := TRUE;
   Ax1_DB2_490 := TRUE;
   Ax2_DB2_492 := TRUE;
   Ax3_DB2_494 := TRUE;
   Ax4_DB2_496 := TRUE;
   Ax5_DB2_498 := TRUE;
   Ax6_DB2_500 := TRUE;
   Ax7_DB2_502 := TRUE;
   Ax8_DB2_504 := TRUE;
   Ax9_DB2_506 := TRUE;
   Ax10_DB2_508 := TRUE;
   Ax11_DB2_510 := TRUE;
   Ax12_DB2_512 := TRUE;
   Ax13_DB2_514 := TRUE;
   Ax14_DB2_516 := TRUE;
   Ax15_DB2_518 := TRUE;
   Ax16_DB2_520 := TRUE;
   Ax17_DB2_522 := TRUE;
   Ax18_DB2_524 := TRUE;
   Ax19_DB2_526 := TRUE;
   Ax20_DB2_528 := TRUE;
   Ax21_DB2_530 := TRUE;
   Ax22_DB2_532 := TRUE;
   Ax23_DB2_534 := TRUE;
   Ax24_DB2_536 := TRUE;
   Ax25_DB2_538 := TRUE;
   Ax26_DB2_540 := TRUE;
   Ax27_DB2_542 := TRUE;
   Ax28_DB2_544 := TRUE;
   Ax29_DB2_546 := TRUE;
   Ax30_DB2_548 := TRUE;
   Ax31_DB2_550 := TRUE;
   Ax32_DB2_552 := TRUE;
   User0_DB2_554 := TRUE;
   User0_DB2_555 := TRUE;
   User0_DB2_556 := TRUE;
   User0_DB2_557 := TRUE;
   User1_DB2_562 := TRUE;
   User1_DB2_563 := TRUE;
   User1_DB2_564 := TRUE;
   User1_DB2_565 := TRUE;
   User2_DB2_570 := TRUE;
   User2_DB2_571 := TRUE;
   User2_DB2_572 := TRUE;
   User2_DB2_573 := TRUE;
   User3_DB2_578 := TRUE;
   User3_DB2_579 := TRUE;
   User3_DB2_580 := TRUE;
   User3_DB2_581 := TRUE;
   User4_DB2_586 := TRUE;
   User4_DB2_587 := TRUE;
   User4_DB2_588 := TRUE;
   User4_DB2_589 := TRUE;
   User5_DB2_594 := TRUE;
   User5_DB2_595 := TRUE;
   User5_DB2_596 := TRUE;
   User5_DB2_597 := TRUE;
   User6_DB2_602 := TRUE;
   User6_DB2_603 := TRUE;
   User6_DB2_604 := TRUE;
   User6_DB2_605 := TRUE;
   User7_DB2_610 := TRUE;
   User7_DB2_611 := TRUE;
   User7_DB2_612 := TRUE;
   User7_DB2_613 := TRUE;
   User8_DB2_618 := TRUE;
   User8_DB2_619 := TRUE;
   User8_DB2_620 := TRUE;
   User8_DB2_621 := TRUE;
   User9_DB2_626 := TRUE;
   User9_DB2_627 := TRUE;
   User9_DB2_628 := TRUE;
   User9_DB2_629 := TRUE;
   User10_DB2_634 := TRUE;
   User10_DB2_635 := TRUE;
   User10_DB2_636 := TRUE;
   User10_DB2_637 := TRUE;
   User11_DB2_642 := TRUE;
   User11_DB2_643 := TRUE;
   User11_DB2_644 := TRUE;
   User11_DB2_645 := TRUE;
   User12_DB2_650 := TRUE;
   User12_DB2_651 := TRUE;
   User12_DB2_652 := TRUE;
   User12_DB2_653 := TRUE;
   User13_DB2_658 := TRUE;
   User13_DB2_659 := TRUE;
   User13_DB2_660 := TRUE;
   User13_DB2_661 := TRUE;
   User14_DB2_666 := TRUE;
   User14_DB2_667 := TRUE;
   User14_DB2_668 := TRUE;
   User14_DB2_669 := TRUE;
   User15_DB2_674 := TRUE;
   User15_DB2_675 := TRUE;
   User15_DB2_676 := TRUE;
   User15_DB2_677 := TRUE;
   User16_DB2_682 := TRUE;
   User16_DB2_683 := TRUE;
   User16_DB2_684 := TRUE;
   User16_DB2_685 := TRUE;
   User17_DB2_690 := TRUE;
   User17_DB2_691 := TRUE;
   User17_DB2_692 := TRUE;
   User17_DB2_693 := TRUE;
   User18_DB2_698 := TRUE;
   User18_DB2_699 := TRUE;
   User18_DB2_700 := TRUE;
   User18_DB2_701 := TRUE;
   User19_DB2_706 := TRUE;
   User19_DB2_707 := TRUE;
   User19_DB2_708 := TRUE;
   User19_DB2_709 := TRUE;
   User20_DB2_714 := TRUE;
   User20_DB2_715 := TRUE;
   User20_DB2_716 := TRUE;
   User20_DB2_717 := TRUE;
   User21_DB2_722 := TRUE;
   User21_DB2_723 := TRUE;
   User21_DB2_724 := TRUE;
   User21_DB2_725 := TRUE;
   User22_DB2_730 := TRUE;
   User22_DB2_731 := TRUE;
   User22_DB2_732 := TRUE;
   User22_DB2_733 := TRUE;
   User23_DB2_738 := TRUE;
   User23_DB2_739 := TRUE;
   User23_DB2_740 := TRUE;
   User23_DB2_741 := TRUE;
   User24_DB2_746 := TRUE;
   User24_DB2_747 := TRUE;
   User24_DB2_748 := TRUE;
   User24_DB2_749 := TRUE;
   User25_DB2_754 := TRUE;
   User25_DB2_755 := TRUE;
   User25_DB2_756 := TRUE;
   User25_DB2_757 := TRUE;
   User26_DB2_762 := TRUE;
   User26_DB2_763 := TRUE;
   User26_DB2_764 := TRUE;
   User26_DB2_765 := TRUE;
   User27_DB2_770 := TRUE;
   User27_DB2_771 := TRUE;
   User27_DB2_772 := TRUE;
   User27_DB2_773 := TRUE;
   User28_DB2_778 := TRUE;
   User28_DB2_779 := TRUE;
   User28_DB2_780 := TRUE;
   User28_DB2_781 := TRUE;
   User29_DB2_786 := TRUE;
   User29_DB2_787 := TRUE;
   User29_DB2_788 := TRUE;
   User29_DB2_789 := TRUE;
   User30_DB2_794 := TRUE;
   User30_DB2_795 := TRUE;
   User30_DB2_796 := TRUE;
   User30_DB2_797 := TRUE;
   User31_DB2_802 := TRUE;
   User31_DB2_803 := TRUE;
   User31_DB2_804 := TRUE;
   User31_DB2_805 := TRUE;
END_DATA_BLOCK

DATA_BLOCK "gp_par"	// DB 7
TITLE = Parameters for Baseprogram
AUTHOR : NUMERIK
FAMILY : _800D
NAME : Basics
VERSION : 2.7
"RUN_UP"
BEGIN
END_DATA_BLOCK

